LIN {X 0,Y 528.073,Z 998.814,A -85,B 0,C 180,E1 -10169.241,E2 -10169.241} C_VEL
LIN {X 0,Y 528.091,Z 998.55,A -85,B 0,C 180,E1 -10171.628,E2 -10171.628} C_VEL
LIN {X 0,Y 528.095,Z 996.5,A -85,B 0,C 180,E1 -10174.235,E2 -10174.235} C_VEL
LIN {X 0,Y 528.112,Z 993.292,A -85,B 0,C 180,E1 -10176.523,E2 -10176.523} C_VEL
LIN {X 0,Y 528.202,Z 987.95,A -85,B 0,C 180,E1 -10179.15,E2 -10179.15} C_VEL
LIN {X 0,Y 528.409,Z 981.754,A -85,B 0,C 180,E1 -10181.421,E2 -10181.421} C_VEL
LIN {X 0,Y 528.804,Z 973.873,A -85,B 0,C 180,E1 -10183.783,E2 -10183.783} C_VEL
LIN {X 0,Y 529.458,Z 963.843,A -85,B 0,C 180,E1 -10186.23,E2 -10186.23} C_VEL
LIN {X 0,Y 530.258,Z 953.621,A -85,B 0,C 180,E1 -10188.355,E2 -10188.355} C_VEL
LIN {X 0,Y 531.541,Z 939.728,A -85,B 0,C 180,E1 -10190.826,E2 -10190.826} C_VEL
LIN {X 0,Y 532.919,Z 926.263,A -85,B 0,C 180,E1 -10192.891,E2 -10192.891} C_VEL
LIN {X 0,Y 534.753,Z 909.549,A -85,B 0,C 180,E1 -10195.116,E2 -10195.116} C_VEL
LIN {X 0,Y 536.55,Z 894.005,A -85,B 0,C 180,E1 -10196.926,E2 -10196.926} C_VEL
LIN {X 0,Y 538.909,Z 873.935,A -85,B 0,C 180,E1 -10198.964,E2 -10198.964} C_VEL
LIN {X 0,Y 541.194,Z 854.701,A -85,B 0,C 180,E1 -10200.659,E2 -10200.659} C_VEL
LIN {X 0,Y 543.603,Z 833.893,A -85,B 0,C 180,E1 -10202.237,E2 -10202.237} C_VEL
LIN {X 0,Y 545.862,Z 813.459,A -85,B 0,C 180,E1 -10203.586,E2 -10203.586} C_VEL
LIN {X 0,Y 548.077,Z 791.418,A -85,B 0,C 180,E1 -10204.822,E2 -10204.822} C_VEL
LIN {X 0,Y 550.284,Z 768.641,A -85,B 0,C 180,E1 -10205.902,E2 -10205.902} C_VEL
LIN {X 0,Y 552.167,Z 745.38,A -85,B 0,C 180,E1 -10206.794,E2 -10206.794} C_VEL
LIN {X 0,Y 553.867,Z 721.472,A -85,B 0,C 180,E1 -10207.53,E2 -10207.53} C_VEL
LIN {X 0,Y 555.081,Z 698.627,A -85,B 0,C 180,E1 -10208.055,E2 -10208.055} C_VEL
LIN {X 0,Y 556.026,Z 670.252,A -85,B 0,C 180,E1 -10208.516,E2 -10208.516} C_VEL
LIN {X 0,Y 558.703,Z 568.517,A -85,B 0,C 180,E1 -10210.011,E2 -10210.011} C_VEL
LIN {X 0,Y 562.298,Z 475.68,A -85,B 0,C 180,E1 -10211.53,E2 -10211.53} C_VEL
LIN {X 0,Y 567.172,Z 389.799,A -85,B 0,C 180,E1 -10213.068,E2 -10213.068} C_VEL
LIN {X 0,Y 570.884,Z 340.567,A -85,B 0,C 180,E1 -10214.019,E2 -10214.019} C_VEL
LIN {X 0,Y 571.881,Z 338.159,A -85,B 0,C 180,E1 -10214.167,E2 -10214.167} C_VEL
LIN {X 0,Y 579.094,Z 319.344,A -85,B 0,C 180,E1 -10215.771,E2 -10215.771} C_VEL
LIN {X 0,Y 582.937,Z 311.16,A -85,B 0,C 180,E1 -10216.542,E2 -10216.542} C_VEL
LIN {X 0,Y 582.832,Z 309.162,A -85,B 0,C 180,E1 -10217.606,E2 -10217.606} C_VEL
LIN {X 0,Y 582.89,Z 308.585,A -85,B 0,C 180,E1 -10218.273,E2 -10218.273} C_VEL
LIN {X 0,Y 582.338,Z 310.355,A -85,B 0,C 180,E1 -10219.595,E2 -10219.595} C_VEL
LIN {X 0,Y 574.337,Z 326.452,A -85,B 0,C 180,E1 -10221.318,E2 -10221.318} C_VEL
LIN {X 0,Y 566.735,Z 346.819,A -85,B 0,C 180,E1 -10223.329,E2 -10223.329} C_VEL
LIN {X 0,Y 559.494,Z 373.809,A -85,B 0,C 180,E1 -10225.802,E2 -10225.802} C_VEL
LIN {X 0,Y 554.301,Z 400.115,A -85,B 0,C 180,E1 -10228.04,E2 -10228.04} C_VEL
LIN {X 0,Y 555.519,Z 423.333,A -85,B 0,C 180,E1 -10229.307,E2 -10229.307} C_VEL
LIN {X 0,Y 556.922,Z 451.305,A -85,B 0,C 180,E1 -10230.635,E2 -10230.635} C_VEL
LIN {X 0,Y 558.184,Z 484.283,A -85,B 0,C 180,E1 -10231.98,E2 -10231.98} C_VEL
LIN {X 0,Y 558.47,Z 501.799,A -85,B 0,C 180,E1 -10232.6,E2 -10232.6} C_VEL
LIN {X 0,Y 549.884,Z 603.402,A -85,B 0,C 180,E1 -10234.933,E2 -10234.933} C_VEL
LIN {X 0,Y 544.198,Z 689.935,A -85,B 0,C 180,E1 -10236.896,E2 -10236.896} C_VEL
LIN {X 0,Y 542.555,Z 713.994,A -85,B 0,C 180,E1 -10237.66,E2 -10237.66} C_VEL
LIN {X 0,Y 541.005,Z 736.005,A -85,B 0,C 180,E1 -10238.568,E2 -10238.568} C_VEL
LIN {X 0,Y 539.398,Z 756.989,A -85,B 0,C 180,E1 -10239.661,E2 -10239.661} C_VEL
LIN {X 0,Y 538.011,Z 774.87,A -85,B 0,C 180,E1 -10240.795,E2 -10240.795} C_VEL
LIN {X 0,Y 536.611,Z 791.893,A -85,B 0,C 180,E1 -10242.094,E2 -10242.094} C_VEL
LIN {X 0,Y 535.34,Z 806.843,A -85,B 0,C 180,E1 -10243.451,E2 -10243.451} C_VEL
LIN {X 0,Y 534.145,Z 820.367,A -85,B 0,C 180,E1 -10244.918,E2 -10244.918} C_VEL
LIN {X 0,Y 533.023,Z 832.916,A -85,B 0,C 180,E1 -10246.549,E2 -10246.549} C_VEL
LIN {X 0,Y 532.018,Z 843.847,A -85,B 0,C 180,E1 -10248.289,E2 -10248.289} C_VEL
LIN {X 0,Y 531.163,Z 853.18,A -85,B 0,C 180,E1 -10250.136,E2 -10250.136} C_VEL
LIN {X 0,Y 530.507,Z 860.457,A -85,B 0,C 180,E1 -10251.983,E2 -10251.983} C_VEL
LIN {X 0,Y 530,Z 866.128,A -85,B 0,C 180,E1 -10253.935,E2 -10253.935} C_VEL
LIN {X 0,Y 529.624,Z 869.937,A -85,B 0,C 180,E1 -10255.886,E2 -10255.886} C_VEL
LIN {X 0,Y 529.372,Z 871.943,A -85,B 0,C 180,E1 -10257.835,E2 -10257.835} C_VEL
LIN {X 0,Y 529.209,Z 872.179,A -85,B 0,C 180,E1 -10259.892,E2 -10259.892} C_VEL
LIN {X 0,Y 529.126,Z 870.512,A -85,B 0,C 180,E1 -10261.949,E2 -10261.949} C_VEL
LIN {X 0,Y 529.146,Z 867.199,A -85,B 0,C 180,E1 -10263.901,E2 -10263.901} C_VEL
LIN {X 0,Y 529.276,Z 862.125,A -85,B 0,C 180,E1 -10265.855,E2 -10265.855} C_VEL
LIN {X 0,Y 529.52,Z 855.186,A -85,B 0,C 180,E1 -10267.814,E2 -10267.814} C_VEL
LIN {X 0,Y 529.941,Z 846.185,A -85,B 0,C 180,E1 -10269.777,E2 -10269.777} C_VEL
LIN {X 0,Y 530.543,Z 835.567,A -85,B 0,C 180,E1 -10271.634,E2 -10271.634} C_VEL
LIN {X 0,Y 531.311,Z 823.375,A -85,B 0,C 180,E1 -10273.384,E2 -10273.384} C_VEL
LIN {X 0,Y 532.271,Z 809.122,A -85,B 0,C 180,E1 -10275.079,E2 -10275.079} C_VEL
LIN {X 0,Y 533.351,Z 793.597,A -85,B 0,C 180,E1 -10276.613,E2 -10276.613} C_VEL
LIN {X 0,Y 534.503,Z 776.998,A -85,B 0,C 180,E1 -10277.979,E2 -10277.979} C_VEL
LIN {X 0,Y 535.659,Z 759.422,A -85,B 0,C 180,E1 -10279.18,E2 -10279.18} C_VEL
LIN {X 0,Y 536.845,Z 740.956,A -85,B 0,C 180,E1 -10280.212,E2 -10280.212} C_VEL
LIN {X 0,Y 537.985,Z 720.972,A -85,B 0,C 180,E1 -10281.106,E2 -10281.106} C_VEL
LIN {X 0,Y 538.984,Z 700.182,A -85,B 0,C 180,E1 -10281.812,E2 -10281.812} C_VEL
LIN {X 0,Y 539.819,Z 679.295,A -85,B 0,C 180,E1 -10282.316,E2 -10282.316} C_VEL
LIN {X 0,Y 545.343,Z 494.327,A -85,B 0,C 180,E1 -10285.454,E2 -10285.454} C_VEL
LIN {X 0,Y 540.838,Z 450.424,A -85,B 0,C 180,E1 -10286.544,E2 -10286.544} C_VEL
LIN {X 0,Y 544.277,Z 398.054,A -85,B 0,C 180,E1 -10290.14,E2 -10290.14} C_VEL
LIN {X 0,Y 547.874,Z 348.579,A -85,B 0,C 180,E1 -10293.572,E2 -10293.572} C_VEL
LIN {X 0,Y 552.064,Z 296.542,A -85,B 0,C 180,E1 -10297.224,E2 -10297.224} C_VEL
LIN {X 0,Y 553.399,Z 279.163,A -85,B 0,C 180,E1 -10298.468,E2 -10298.468} C_VEL
LIN {X 0,Y 544.537,Z 255.5,A -85,B 0,C 180,E1 -10301.002,E2 -10301.002} C_VEL
LIN {X 0,Y 535.075,Z 232.411,A -85,B 0,C 180,E1 -10303.682,E2 -10303.682} C_VEL
LIN {X 0,Y 534.781,Z 231.7,A -85,B 0,C 180,E1 -10303.773,E2 -10303.773} C_VEL
LIN {X 0,Y 536.691,Z 232.864,A -85,B 0,C 180,E1 -10304.059,E2 -10304.059} C_VEL
LIN {X 0,Y 546.06,Z 252.219,A -85,B 0,C 180,E1 -10306.403,E2 -10306.403} C_VEL
LIN {X 0,Y 554.586,Z 272.537,A -85,B 0,C 180,E1 -10308.749,E2 -10308.749} C_VEL
LIN {X 0,Y 561.348,Z 291.078,A -85,B 0,C 180,E1 -10310.79,E2 -10310.79} C_VEL
LIN {X 0,Y 561.17,Z 298.745,A -85,B 0,C 180,E1 -10311.342,E2 -10311.342} C_VEL
LIN {X 0,Y 560.235,Z 305.401,A -85,B 0,C 180,E1 -10311.739,E2 -10311.739} C_VEL
LIN {X 0,Y 555.035,Z 324.312,A -85,B 0,C 180,E1 -10312.584,E2 -10312.584} C_VEL
LIN {X 0,Y 554.398,Z 330.093,A -85,B 0,C 180,E1 -10312.919,E2 -10312.919} C_VEL
LIN {X 0,Y 554.416,Z 348.963,A -85,B 0,C 180,E1 -10314.148,E2 -10314.148} C_VEL
LIN {X 0,Y 552.164,Z 359.982,A -85,B 0,C 180,E1 -10314.558,E2 -10314.558} C_VEL
LIN {X 0,Y 549.54,Z 449.417,A -85,B 0,C 180,E1 -10315.862,E2 -10315.862} C_VEL
LIN {X 0,Y 546.257,Z 527.382,A -85,B 0,C 180,E1 -10317.185,E2 -10317.185} C_VEL
LIN {X 0,Y 541.758,Z 616.567,A -85,B 0,C 180,E1 -10318.913,E2 -10318.913} C_VEL
LIN {X 0,Y 540.542,Z 646.224,A -85,B 0,C 180,E1 -10319.6,E2 -10319.6} C_VEL
LIN {X 0,Y 539.38,Z 668.071,A -85,B 0,C 180,E1 -10320.302,E2 -10320.302} C_VEL
LIN {X 0,Y 537.858,Z 689.945,A -85,B 0,C 180,E1 -10321.217,E2 -10321.217} C_VEL
LIN {X 0,Y 536.147,Z 710.107,A -85,B 0,C 180,E1 -10322.27,E2 -10322.27} C_VEL
LIN {X 0,Y 534.288,Z 729.488,A -85,B 0,C 180,E1 -10323.491,E2 -10323.491} C_VEL
LIN {X 0,Y 532.25,Z 748.721,A -85,B 0,C 180,E1 -10324.936,E2 -10324.936} C_VEL
LIN {X 0,Y 530.139,Z 767.337,A -85,B 0,C 180,E1 -10326.597,E2 -10326.597} C_VEL
LIN {X 0,Y 528.194,Z 784.001,A -85,B 0,C 180,E1 -10328.355,E2 -10328.355} C_VEL
LIN {X 0,Y 526.509,Z 798.406,A -85,B 0,C 180,E1 -10330.127,E2 -10330.127} C_VEL
LIN {X 0,Y 524.913,Z 812.343,A -85,B 0,C 180,E1 -10332.14,E2 -10332.14} C_VEL
LIN {X 0,Y 523.561,Z 824.713,A -85,B 0,C 180,E1 -10334.268,E2 -10334.268} C_VEL
LIN {X 0,Y 522.516,Z 835.264,A -85,B 0,C 180,E1 -10336.438,E2 -10336.438} C_VEL
LIN {X 0,Y 521.742,Z 844.408,A -85,B 0,C 180,E1 -10338.727,E2 -10338.727} C_VEL
LIN {X 0,Y 521.227,Z 851.534,A -85,B 0,C 180,E1 -10340.949,E2 -10340.949} C_VEL
LIN {X 0,Y 520.916,Z 857.237,A -85,B 0,C 180,E1 -10343.276,E2 -10343.276} C_VEL
LIN {X 0,Y 520.738,Z 861.151,A -85,B 0,C 180,E1 -10345.595,E2 -10345.595} C_VEL
LIN {X 0,Y 520.657,Z 863.456,A -85,B 0,C 180,E1 -10347.909,E2 -10347.909} C_VEL
LIN {X 0,Y 520.639,Z 864.185,A -85,B 0,C 180,E1 -10350.22,E2 -10350.22} C_VEL
LIN {X 0,Y 520.658,Z 863.243,A -85,B 0,C 180,E1 -10352.532,E2 -10352.532} C_VEL
LIN {X 0,Y 520.758,Z 860.648,A -85,B 0,C 180,E1 -10354.846,E2 -10354.846} C_VEL
LIN {X 0,Y 520.942,Z 856.196,A -85,B 0,C 180,E1 -10357.278,E2 -10357.278} C_VEL
LIN {X 0,Y 521.293,Z 850.544,A -85,B 0,C 180,E1 -10359.495,E2 -10359.495} C_VEL
LIN {X 0,Y 521.889,Z 842.757,A -85,B 0,C 180,E1 -10361.83,E2 -10361.83} C_VEL
LIN {X 0,Y 522.691,Z 833.442,A -85,B 0,C 180,E1 -10364.06,E2 -10364.06} C_VEL
LIN {X 0,Y 523.79,Z 822.558,A -85,B 0,C 180,E1 -10366.217,E2 -10366.217} C_VEL
LIN {X 0,Y 525.167,Z 809.983,A -85,B 0,C 180,E1 -10368.31,E2 -10368.31} C_VEL
LIN {X 0,Y 526.732,Z 796.54,A -85,B 0,C 180,E1 -10370.212,E2 -10370.212} C_VEL
LIN {X 0,Y 528.506,Z 781.567,A -85,B 0,C 180,E1 -10372.021,E2 -10372.021} C_VEL
LIN {X 0,Y 530.475,Z 764.694,A -85,B 0,C 180,E1 -10373.753,E2 -10373.753} C_VEL
LIN {X 0,Y 532.444,Z 747.087,A -85,B 0,C 180,E1 -10375.292,E2 -10375.292} C_VEL
LIN {X 0,Y 534.424,Z 728.325,A -85,B 0,C 180,E1 -10376.682,E2 -10376.682} C_VEL
LIN {X 0,Y 536.282,Z 708.692,A -85,B 0,C 180,E1 -10377.904,E2 -10377.904} C_VEL
LIN {X 0,Y 537.972,Z 688.594,A -85,B 0,C 180,E1 -10378.938,E2 -10378.938} C_VEL
LIN {X 0,Y 539.445,Z 667.47,A -85,B 0,C 180,E1 -10379.815,E2 -10379.815} C_VEL
LIN {X 0,Y 540.613,Z 645.234,A -85,B 0,C 180,E1 -10380.523,E2 -10380.523} C_VEL
LIN {X 0,Y 541.962,Z 612.731,A -85,B 0,C 180,E1 -10381.262,E2 -10381.262} C_VEL
LIN {X 0,Y 546.474,Z 523.52,A -85,B 0,C 180,E1 -10382.98,E2 -10382.98} C_VEL
LIN {X 0,Y 549.681,Z 446.416,A -85,B 0,C 180,E1 -10384.279,E2 -10384.279} C_VEL
LIN {X 0,Y 552.294,Z 358.711,A -85,B 0,C 180,E1 -10385.563,E2 -10385.563} C_VEL
LIN {X 0,Y 554.559,Z 348.099,A -85,B 0,C 180,E1 -10386,E2 -10386} C_VEL
LIN {X 0,Y 554.663,Z 312.521,A -85,B 0,C 180,E1 -10388.391,E2 -10388.391} C_VEL
LIN {X 0,Y 554.973,Z 294.272,A -85,B 0,C 180,E1 -10389.707,E2 -10389.707} C_VEL
LIN {X 0,Y 547.767,Z 275.074,A -85,B 0,C 180,E1 -10391.861,E2 -10391.861} C_VEL
LIN {X 0,Y 539.853,Z 256.334,A -85,B 0,C 180,E1 -10394.058,E2 -10394.058} C_VEL
LIN {X 0,Y 532.349,Z 240.84,A -85,B 0,C 180,E1 -10395.976,E2 -10395.976} C_VEL
LIN {X 0,Y 526.336,Z 229.281,A -85,B 0,C 180,E1 -10397.445,E2 -10397.445} C_VEL
LIN {X 0,Y 523.694,Z 224.562,A -85,B 0,C 180,E1 -10398.067,E2 -10398.067} C_VEL
LIN {X 0,Y 521.964,Z 221.334,A -85,B 0,C 180,E1 -10398.485,E2 -10398.485} C_VEL
LIN {X 0,Y 521.744,Z 220.235,A -85,B 0,C 180,E1 -10398.61,E2 -10398.61} C_VEL
LIN {X 0,Y 521.743,Z 220.233,A -85,B 0,C 180,E1 -10402.035,E2 -10402.035} C_VEL
LIN {X 0,Y 521.737,Z 220.239,A -85,B 0,C 180,E1 -10405.495,E2 -10405.495} C_VEL
LIN {X 0,Y 521.735,Z 220.239,A -85,B 0,C 180,E1 -10408.967,E2 -10408.967} C_VEL
LIN {X 0,Y 521.739,Z 220.219,A -85,B 0,C 180,E1 -10412.368,E2 -10412.368} C_VEL
LIN {X 0,Y 521.742,Z 220.211,A -85,B 0,C 180,E1 -10415.815,E2 -10415.815} C_VEL
LIN {X 0,Y 521.737,Z 220.238,A -85,B 0,C 180,E1 -10419.266,E2 -10419.266} C_VEL
LIN {X 0,Y 521.741,Z 220.21,A -85,B 0,C 180,E1 -10422.719,E2 -10422.719} C_VEL
LIN {X 0,Y 521.732,Z 220.223,A -85,B 0,C 180,E1 -10426.139,E2 -10426.139} C_VEL
LIN {X 0,Y 521.742,Z 220.225,A -85,B 0,C 180,E1 -10429.622,E2 -10429.622} C_VEL
LIN {X 0,Y 521.745,Z 220.21,A -85,B 0,C 180,E1 -10433.078,E2 -10433.078} C_VEL
LIN {X 0,Y 521.729,Z 220.239,A -85,B 0,C 180,E1 -10436.594,E2 -10436.594} C_VEL
LIN {X 0,Y 521.726,Z 220.202,A -85,B 0,C 180,E1 -10440.11,E2 -10440.11} C_VEL
LIN {X 0,Y 521.744,Z 220.238,A -85,B 0,C 180,E1 -10443.516,E2 -10443.516} C_VEL
LIN {X 0,Y 521.744,Z 220.198,A -85,B 0,C 180,E1 -10447.045,E2 -10447.045} C_VEL
LIN {X 0,Y 521.72,Z 220.241,A -85,B 0,C 180,E1 -10450.524,E2 -10450.524} C_VEL
LIN {X 0,Y 521.739,Z 220.242,A -85,B 0,C 180,E1 -10453.974,E2 -10453.974} C_VEL
LIN {X 0,Y 521.749,Z 220.241,A -85,B 0,C 180,E1 -10457.395,E2 -10457.395} C_VEL
LIN {X 0,Y 521.717,Z 220.239,A -85,B 0,C 180,E1 -10460.767,E2 -10460.767} C_VEL
LIN {X 0,Y 521.722,Z 220.235,A -85,B 0,C 180,E1 -10464.213,E2 -10464.213} C_VEL
LIN {X 0,Y 521.753,Z 220.235,A -85,B 0,C 180,E1 -10467.631,E2 -10467.631} C_VEL
LIN {X 0,Y 521.722,Z 220.239,A -85,B 0,C 180,E1 -10471.054,E2 -10471.054} C_VEL
LIN {X 0,Y 521.754,Z 220.325,A -85,B 0,C 180,E1 -10473.388,E2 -10473.388} C_VEL
LIN {X 0,Y 522.874,Z 223.439,A -85,B 0,C 180,E1 -10473.813,E2 -10473.813} C_VEL
LIN {X 0,Y 524.045,Z 225.27,A -85,B 0,C 180,E1 -10474.122,E2 -10474.122} C_VEL
LIN {X 0,Y 525.794,Z 228.852,A -85,B 0,C 180,E1 -10474.653,E2 -10474.653} C_VEL
LIN {X 0,Y 533.823,Z 244.524,A -85,B 0,C 180,E1 -10476.96,E2 -10476.96} C_VEL
LIN {X 0,Y 543.759,Z 264.219,A -85,B 0,C 180,E1 -10479.649,E2 -10479.649} C_VEL
LIN {X 0,Y 556.286,Z 289.963,A -85,B 0,C 180,E1 -10482.832,E2 -10482.832} C_VEL
LIN {X 0,Y 561.303,Z 300.628,A -85,B 0,C 180,E1 -10484.054,E2 -10484.054} C_VEL
LIN {X 0,Y 559.967,Z 313.808,A -85,B 0,C 180,E1 -10484.827,E2 -10484.827} C_VEL
LIN {X 0,Y 562.81,Z 340.382,A -85,B 0,C 180,E1 -10485.543,E2 -10485.543} C_VEL
LIN {X 0,Y 554.944,Z 572.433,A -85,B 0,C 180,E1 -10489.082,E2 -10489.082} C_VEL
LIN {X 0,Y 551.384,Z 692.781,A -85,B 0,C 180,E1 -10490.881,E2 -10490.881} C_VEL
LIN {X 0,Y 549.935,Z 717.309,A -85,B 0,C 180,E1 -10491.421,E2 -10491.421} C_VEL
LIN {X 0,Y 548.22,Z 740.807,A -85,B 0,C 180,E1 -10492.107,E2 -10492.107} C_VEL
LIN {X 0,Y 546.127,Z 763.625,A -85,B 0,C 180,E1 -10492.965,E2 -10492.965} C_VEL
LIN {X 0,Y 543.758,Z 786.648,A -85,B 0,C 180,E1 -10494.008,E2 -10494.008} C_VEL
LIN {X 0,Y 541.136,Z 809.081,A -85,B 0,C 180,E1 -10495.247,E2 -10495.247} C_VEL
LIN {X 0,Y 538.432,Z 830.883,A -85,B 0,C 180,E1 -10496.655,E2 -10496.655} C_VEL
LIN {X 0,Y 535.859,Z 850.246,A -85,B 0,C 180,E1 -10498.125,E2 -10498.125} C_VEL
LIN {X 0,Y 533.106,Z 870.475,A -85,B 0,C 180,E1 -10499.886,E2 -10499.886} C_VEL
LIN {X 0,Y 530.656,Z 888,A -85,B 0,C 180,E1 -10501.652,E2 -10501.652} C_VEL
LIN {X 0,Y 528.37,Z 904.978,A -85,B 0,C 180,E1 -10503.595,E2 -10503.595} C_VEL
LIN {X 0,Y 526.295,Z 920.525,A -85,B 0,C 180,E1 -10505.652,E2 -10505.652} C_VEL
LIN {X 0,Y 524.481,Z 935.456,A -85,B 0,C 180,E1 -10507.901,E2 -10507.901} C_VEL
LIN {X 0,Y 523.037,Z 948.215,A -85,B 0,C 180,E1 -10510.146,E2 -10510.146} C_VEL
LIN {X 0,Y 521.869,Z 960.375,A -85,B 0,C 180,E1 -10512.609,E2 -10512.609} C_VEL
LIN {X 0,Y 521.085,Z 970.191,A -85,B 0,C 180,E1 -10514.987,E2 -10514.987} C_VEL
LIN {X 0,Y 520.553,Z 978.856,A -85,B 0,C 180,E1 -10517.464,E2 -10517.464} C_VEL
LIN {X 0,Y 520.257,Z 985.967,A -85,B 0,C 180,E1 -10520.039,E2 -10520.039} C_VEL
LIN {X 0,Y 520.116,Z 990.812,A -85,B 0,C 180,E1 -10522.266,E2 -10522.266} C_VEL
LIN {X 0,Y 520.085,Z 994.867,A -85,B 0,C 180,E1 -10524.816,E2 -10524.816} C_VEL
LIN {X 0,Y 520.101,Z 997.064,A -85,B 0,C 180,E1 -10527.135,E2 -10527.135} C_VEL
LIN {X 0,Y 520.12,Z 997.946,A -85,B 0,C 180,E1 -10529.229,E2 -10529.229} C_VEL
LIN {X 0,Y 520.139,Z 997.696,A -85,B 0,C 180,E1 -10531.561,E2 -10531.561} C_VEL
LIN {X 0,Y 520.139,Z 995.709,A -85,B 0,C 180,E1 -10534.189,E2 -10534.189} C_VEL
LIN {X 0,Y 520.149,Z 992.525,A -85,B 0,C 180,E1 -10536.512,E2 -10536.512} C_VEL
LIN {X 0,Y 520.233,Z 987.22,A -85,B 0,C 180,E1 -10539.18,E2 -10539.18} C_VEL
LIN {X 0,Y 520.439,Z 980.92,A -85,B 0,C 180,E1 -10541.526,E2 -10541.526} C_VEL
LIN {X 0,Y 520.81,Z 973.556,A -85,B 0,C 180,E1 -10543.772,E2 -10543.772} C_VEL
LIN {X 0,Y 521.5,Z 963.155,A -85,B 0,C 180,E1 -10546.371,E2 -10546.371} C_VEL
LIN {X 0,Y 522.274,Z 953.521,A -85,B 0,C 180,E1 -10548.415,E2 -10548.415} C_VEL
LIN {X 0,Y 523.524,Z 940.476,A -85,B 0,C 180,E1 -10550.809,E2 -10550.809} C_VEL
LIN {X 0,Y 524.882,Z 927.409,A -85,B 0,C 180,E1 -10552.869,E2 -10552.869} C_VEL
LIN {X 0,Y 526.69,Z 911.753,A -85,B 0,C 180,E1 -10555.047,E2 -10555.047} C_VEL
LIN {X 0,Y 528.751,Z 894.474,A -85,B 0,C 180,E1 -10557.113,E2 -10557.113} C_VEL
LIN {X 0,Y 531.057,Z 875.875,A -85,B 0,C 180,E1 -10559.063,E2 -10559.063} C_VEL
LIN {X 0,Y 533.395,Z 856.932,A -85,B 0,C 180,E1 -10560.781,E2 -10560.781} C_VEL
LIN {X 0,Y 536.068,Z 835.167,A -85,B 0,C 180,E1 -10562.492,E2 -10562.492} C_VEL
LIN {X 0,Y 538.313,Z 815.895,A -85,B 0,C 180,E1 -10563.801,E2 -10563.801} C_VEL
LIN {X 0,Y 540.838,Z 792.483,A -85,B 0,C 180,E1 -10565.162,E2 -10565.162} C_VEL
LIN {X 0,Y 543.143,Z 769.878,A -85,B 0,C 180,E1 -10566.261,E2 -10566.261} C_VEL
LIN {X 0,Y 545.171,Z 746.679,A -85,B 0,C 180,E1 -10567.181,E2 -10567.181} C_VEL
LIN {X 0,Y 546.946,Z 723.653,A -85,B 0,C 180,E1 -10567.919,E2 -10567.919} C_VEL
LIN {X 0,Y 548.337,Z 699.785,A -85,B 0,C 180,E1 -10568.49,E2 -10568.49} C_VEL
LIN {X 0,Y 549.321,Z 674.5,A -85,B 0,C 180,E1 -10568.926,E2 -10568.926} C_VEL
LIN {X 0,Y 552.201,Z 576.067,A -85,B 0,C 180,E1 -10570.412,E2 -10570.412} C_VEL
LIN {X 0,Y 556.018,Z 486.791,A -85,B 0,C 180,E1 -10571.912,E2 -10571.912} C_VEL
LIN {X 0,Y 561.161,Z 403.595,A -85,B 0,C 180,E1 -10573.442,E2 -10573.442} C_VEL
LIN {X 0,Y 566.111,Z 343.623,A -85,B 0,C 180,E1 -10574.63,E2 -10574.63} C_VEL
LIN {X 0,Y 567.547,Z 340.563,A -85,B 0,C 180,E1 -10574.806,E2 -10574.806} C_VEL
LIN {X 0,Y 575.021,Z 323.124,A -85,B 0,C 180,E1 -10576.343,E2 -10576.343} C_VEL
LIN {X 0,Y 578.257,Z 316.88,A -85,B 0,C 180,E1 -10576.934,E2 -10576.934} C_VEL
LIN {X 0,Y 578.346,Z 315.09,A -85,B 0,C 180,E1 -10578.172,E2 -10578.172} C_VEL
LIN {X 0,Y 577.731,Z 316.371,A -85,B 0,C 180,E1 -10579.238,E2 -10579.238} C_VEL
LIN {X 0,Y 568.969,Z 332.766,A -85,B 0,C 180,E1 -10581.013,E2 -10581.013} C_VEL
LIN {X 0,Y 561.23,Z 352.221,A -85,B 0,C 180,E1 -10582.973,E2 -10582.973} C_VEL
LIN {X 0,Y 553.999,Z 376.806,A -85,B 0,C 180,E1 -10585.289,E2 -10585.289} C_VEL
LIN {X 0,Y 549.797,Z 396.074,A -85,B 0,C 180,E1 -10586.972,E2 -10586.972} C_VEL
LIN {X 0,Y 550.632,Z 420.862,A -85,B 0,C 180,E1 -10588.423,E2 -10588.423} C_VEL
LIN {X 0,Y 551.732,Z 450.81,A -85,B 0,C 180,E1 -10589.92,E2 -10589.92} C_VEL
LIN {X 0,Y 552.582,Z 483.66,A -85,B 0,C 180,E1 -10591.317,E2 -10591.317} C_VEL
LIN {X 0,Y 552.788,Z 503.004,A -85,B 0,C 180,E1 -10592.031,E2 -10592.031} C_VEL
LIN {X 0,Y 543.196,Z 609.107,A -85,B 0,C 180,E1 -10594.537,E2 -10594.537} C_VEL
LIN {X 0,Y 537.537,Z 689.387,A -85,B 0,C 180,E1 -10596.414,E2 -10596.414} C_VEL
LIN {X 0,Y 535.83,Z 712.83,A -85,B 0,C 180,E1 -10597.161,E2 -10597.161} C_VEL
LIN {X 0,Y 534.14,Z 734.712,A -85,B 0,C 180,E1 -10598.071,E2 -10598.071} C_VEL
LIN {X 0,Y 532.54,Z 754.757,A -85,B 0,C 180,E1 -10599.1,E2 -10599.1} C_VEL
LIN {X 0,Y 530.937,Z 773.824,A -85,B 0,C 180,E1 -10600.299,E2 -10600.299} C_VEL
LIN {X 0,Y 529.443,Z 791.217,A -85,B 0,C 180,E1 -10601.615,E2 -10601.615} C_VEL
LIN {X 0,Y 527.95,Z 807.44,A -85,B 0,C 180,E1 -10603.099,E2 -10603.099} C_VEL
LIN {X 0,Y 526.676,Z 821.085,A -85,B 0,C 180,E1 -10604.586,E2 -10604.586} C_VEL
LIN {X 0,Y 525.456,Z 833.65,A -85,B 0,C 180,E1 -10606.24,E2 -10606.24} C_VEL
LIN {X 0,Y 524.372,Z 844.771,A -85,B 0,C 180,E1 -10608.017,E2 -10608.017} C_VEL
LIN {X 0,Y 523.445,Z 854.084,A -85,B 0,C 180,E1 -10609.878,E2 -10609.878} C_VEL
LIN {X 0,Y 522.727,Z 861.417,A -85,B 0,C 180,E1 -10611.752,E2 -10611.752} C_VEL
LIN {X 0,Y 522.168,Z 867.158,A -85,B 0,C 180,E1 -10613.734,E2 -10613.734} C_VEL
LIN {X 0,Y 521.752,Z 870.983,A -85,B 0,C 180,E1 -10615.714,E2 -10615.714} C_VEL
LIN {X 0,Y 521.458,Z 873.086,A -85,B 0,C 180,E1 -10617.802,E2 -10617.802} C_VEL
LIN {X 0,Y 521.288,Z 873.282,A -85,B 0,C 180,E1 -10619.78,E2 -10619.78} C_VEL
LIN {X 0,Y 521.191,Z 871.638,A -85,B 0,C 180,E1 -10621.869,E2 -10621.869} C_VEL
LIN {X 0,Y 521.209,Z 868.088,A -85,B 0,C 180,E1 -10623.96,E2 -10623.96} C_VEL
LIN {X 0,Y 521.345,Z 862.924,A -85,B 0,C 180,E1 -10625.945,E2 -10625.945} C_VEL
LIN {X 0,Y 521.604,Z 855.883,A -85,B 0,C 180,E1 -10627.933,E2 -10627.933} C_VEL
LIN {X 0,Y 522.02,Z 847.345,A -85,B 0,C 180,E1 -10629.815,E2 -10629.815} C_VEL
LIN {X 0,Y 522.64,Z 836.731,A -85,B 0,C 180,E1 -10631.7,E2 -10631.7} C_VEL
LIN {X 0,Y 523.432,Z 824.547,A -85,B 0,C 180,E1 -10633.477,E2 -10633.477} C_VEL
LIN {X 0,Y 524.389,Z 810.796,A -85,B 0,C 180,E1 -10635.143,E2 -10635.143} C_VEL
LIN {X 0,Y 525.493,Z 795.428,A -85,B 0,C 180,E1 -10636.698,E2 -10636.698} C_VEL
LIN {X 0,Y 526.724,Z 778.299,A -85,B 0,C 180,E1 -10638.139,E2 -10638.139} C_VEL
LIN {X 0,Y 527.917,Z 760.842,A -85,B 0,C 180,E1 -10639.357,E2 -10639.357} C_VEL
LIN {X 0,Y 529.12,Z 742.725,A -85,B 0,C 180,E1 -10640.396,E2 -10640.396} C_VEL
LIN {X 0,Y 530.265,Z 723.546,A -85,B 0,C 180,E1 -10641.284,E2 -10641.284} C_VEL
LIN {X 0,Y 531.332,Z 702.865,A -85,B 0,C 180,E1 -10642.026,E2 -10642.026} C_VEL
LIN {X 0,Y 532.259,Z 681.478,A -85,B 0,C 180,E1 -10642.574,E2 -10642.574} C_VEL
LIN {X 0,Y 538.097,Z 495.341,A -85,B 0,C 180,E1 -10645.799,E2 -10645.799} C_VEL
LIN {X 0,Y 533.475,Z 449.88,A -85,B 0,C 180,E1 -10646.941,E2 -10646.941} C_VEL
LIN {X 0,Y 537.156,Z 396.261,A -85,B 0,C 180,E1 -10650.667,E2 -10650.667} C_VEL
LIN {X 0,Y 540.798,Z 348.675,A -85,B 0,C 180,E1 -10654.007,E2 -10654.007} C_VEL
LIN {X 0,Y 545.201,Z 296.528,A -85,B 0,C 180,E1 -10657.708,E2 -10657.708} C_VEL
LIN {X 0,Y 546.276,Z 282.025,A -85,B 0,C 180,E1 -10658.763,E2 -10658.763} C_VEL
LIN {X 0,Y 537.787,Z 259.311,A -85,B 0,C 180,E1 -10661.229,E2 -10661.229} C_VEL
LIN {X 0,Y 529.445,Z 238.662,A -85,B 0,C 180,E1 -10663.659,E2 -10663.659} C_VEL
LIN {X 0,Y 531.632,Z 239.348,A -85,B 0,C 180,E1 -10663.949,E2 -10663.949} C_VEL
LIN {X 0,Y 539.955,Z 256.58,A -85,B 0,C 180,E1 -10666.084,E2 -10666.084} C_VEL
LIN {X 0,Y 547.54,Z 274.698,A -85,B 0,C 180,E1 -10668.199,E2 -10668.199} C_VEL
LIN {X 0,Y 554.992,Z 294.722,A -85,B 0,C 180,E1 -10670.441,E2 -10670.441} C_VEL
LIN {X 0,Y 554.398,Z 330.093,A -85,B 0,C 180,E1 -10672.919,E2 -10672.919} C_VEL
LIN {X 0,Y 553.581,Z 335.341,A -85,B 0,C 180,E1 -10673.19,E2 -10673.19} C_VEL
LIN {X 0,Y 547.836,Z 351.92,A -85,B 0,C 180,E1 -10673.701,E2 -10673.701} C_VEL
LIN {X 0,Y 545.655,Z 362.546,A -85,B 0,C 180,E1 -10674.097,E2 -10674.097} C_VEL
LIN {X 0,Y 542.944,Z 451.442,A -85,B 0,C 180,E1 -10675.405,E2 -10675.405} C_VEL
LIN {X 0,Y 539.626,Z 527.403,A -85,B 0,C 180,E1 -10676.711,E2 -10676.711} C_VEL
LIN {X 0,Y 535.005,Z 615.09,A -85,B 0,C 180,E1 -10678.434,E2 -10678.434} C_VEL
LIN {X 0,Y 533.624,Z 647.175,A -85,B 0,C 180,E1 -10679.183,E2 -10679.183} C_VEL
LIN {X 0,Y 532.402,Z 669.345,A -85,B 0,C 180,E1 -10679.904,E2 -10679.904} C_VEL
LIN {X 0,Y 530.865,Z 690.529,A -85,B 0,C 180,E1 -10680.802,E2 -10680.802} C_VEL
LIN {X 0,Y 529.086,Z 710.813,A -85,B 0,C 180,E1 -10681.867,E2 -10681.867} C_VEL
LIN {X 0,Y 527.153,Z 730.268,A -85,B 0,C 180,E1 -10683.103,E2 -10683.103} C_VEL
LIN {X 0,Y 525.02,Z 749.549,A -85,B 0,C 180,E1 -10684.567,E2 -10684.567} C_VEL
LIN {X 0,Y 522.942,Z 767.166,A -85,B 0,C 180,E1 -10686.146,E2 -10686.146} C_VEL
LIN {X 0,Y 521.033,Z 782.83,A -85,B 0,C 180,E1 -10687.787,E2 -10687.787} C_VEL
LIN {X 0,Y 519.068,Z 798.679,A -85,B 0,C 180,E1 -10689.739,E2 -10689.739} C_VEL
LIN {X 0,Y 517.376,Z 812.519,A -85,B 0,C 180,E1 -10691.755,E2 -10691.755} C_VEL
LIN {X 0,Y 515.997,Z 824.407,A -85,B 0,C 180,E1 -10693.797,E2 -10693.797} C_VEL
LIN {X 0,Y 514.817,Z 835.488,A -85,B 0,C 180,E1 -10696.064,E2 -10696.064} C_VEL
LIN {X 0,Y 513.987,Z 844.588,A -85,B 0,C 180,E1 -10698.327,E2 -10698.327} C_VEL
LIN {X 0,Y 513.4,Z 851.915,A -85,B 0,C 180,E1 -10700.584,E2 -10700.584} C_VEL
LIN {X 0,Y 513.02,Z 857.723,A -85,B 0,C 180,E1 -10702.947,E2 -10702.947} C_VEL
LIN {X 0,Y 512.827,Z 861.83,A -85,B 0,C 180,E1 -10705.303,E2 -10705.303} C_VEL
LIN {X 0,Y 512.724,Z 864.323,A -85,B 0,C 180,E1 -10707.653,E2 -10707.653} C_VEL
LIN {X 0,Y 512.715,Z 865.211,A -85,B 0,C 180,E1 -10710,E2 -10710} C_VEL
LIN {X 0,Y 512.721,Z 864.377,A -85,B 0,C 180,E1 -10712.347,E2 -10712.347} C_VEL
LIN {X 0,Y 512.823,Z 861.957,A -85,B 0,C 180,E1 -10714.697,E2 -10714.697} C_VEL
LIN {X 0,Y 513.013,Z 857.929,A -85,B 0,C 180,E1 -10717.053,E2 -10717.053} C_VEL
LIN {X 0,Y 513.376,Z 852.172,A -85,B 0,C 180,E1 -10719.416,E2 -10719.416} C_VEL
LIN {X 0,Y 513.959,Z 844.91,A -85,B 0,C 180,E1 -10721.673,E2 -10721.673} C_VEL
LIN {X 0,Y 514.778,Z 835.896,A -85,B 0,C 180,E1 -10723.937,E2 -10723.937} C_VEL
LIN {X 0,Y 515.881,Z 825.52,A -85,B 0,C 180,E1 -10726.091,E2 -10726.091} C_VEL
LIN {X 0,Y 517.236,Z 813.852,A -85,B 0,C 180,E1 -10728.134,E2 -10728.134} C_VEL
LIN {X 0,Y 518.962,Z 799.602,A -85,B 0,C 180,E1 -10730.23,E2 -10730.23} C_VEL
LIN {X 0,Y 520.817,Z 784.56,A -85,B 0,C 180,E1 -10732.104,E2 -10732.104} C_VEL
LIN {X 0,Y 522.772,Z 768.635,A -85,B 0,C 180,E1 -10733.802,E2 -10733.802} C_VEL
LIN {X 0,Y 524.953,Z 750.305,A -85,B 0,C 180,E1 -10735.465,E2 -10735.465} C_VEL
LIN {X 0,Y 527.06,Z 731.305,A -85,B 0,C 180,E1 -10736.919,E2 -10736.919} C_VEL
LIN {X 0,Y 528.977,Z 712.359,A -85,B 0,C 180,E1 -10738.139,E2 -10738.139} C_VEL
LIN {X 0,Y 530.751,Z 692.432,A -85,B 0,C 180,E1 -10739.205,E2 -10739.205} C_VEL
LIN {X 0,Y 532.312,Z 670.851,A -85,B 0,C 180,E1 -10740.132,E2 -10740.132} C_VEL
LIN {X 0,Y 533.516,Z 649.724,A -85,B 0,C 180,E1 -10740.836,E2 -10740.836} C_VEL
LIN {X 0,Y 534.659,Z 622.529,A -85,B 0,C 180,E1 -10741.501,E2 -10741.501} C_VEL
LIN {X 0,Y 539.133,Z 537.667,A -85,B 0,C 180,E1 -10743.193,E2 -10743.193} C_VEL
LIN {X 0,Y 542.511,Z 463.41,A -85,B 0,C 180,E1 -10744.496,E2 -10744.496} C_VEL
LIN {X 0,Y 544.936,Z 390.36,A -85,B 0,C 180,E1 -10745.604,E2 -10745.604} C_VEL
LIN {X 0,Y 545.777,Z 361.482,A -85,B 0,C 180,E1 -10746.021,E2 -10746.021} C_VEL
LIN {X 0,Y 548.279,Z 350.09,A -85,B 0,C 180,E1 -10746.479,E2 -10746.479} C_VEL
LIN {X 0,Y 548.418,Z 314.014,A -85,B 0,C 180,E1 -10748.91,E2 -10748.91} C_VEL
LIN {X 0,Y 548.648,Z 298.086,A -85,B 0,C 180,E1 -10750.054,E2 -10750.054} C_VEL
LIN {X 0,Y 541.116,Z 277.916,A -85,B 0,C 180,E1 -10752.342,E2 -10752.342} C_VEL
LIN {X 0,Y 533.24,Z 259.389,A -85,B 0,C 180,E1 -10754.557,E2 -10754.557} C_VEL
LIN {X 0,Y 524.905,Z 242.374,A -85,B 0,C 180,E1 -10756.704,E2 -10756.704} C_VEL
LIN {X 0,Y 518.482,Z 230.32,A -85,B 0,C 180,E1 -10758.292,E2 -10758.292} C_VEL
LIN {X 0,Y 515.867,Z 225.675,A -85,B 0,C 180,E1 -10758.923,E2 -10758.923} C_VEL
LIN {X 0,Y 514.115,Z 222.681,A -85,B 0,C 180,E1 -10759.342,E2 -10759.342} C_VEL
LIN {X 0,Y 513.798,Z 221.214,A -85,B 0,C 180,E1 -10759.502,E2 -10759.502} C_VEL
LIN {X 0,Y 513.791,Z 221.21,A -85,B 0,C 180,E1 -10763.033,E2 -10763.033} C_VEL
LIN {X 0,Y 513.805,Z 221.208,A -85,B 0,C 180,E1 -10766.449,E2 -10766.449} C_VEL
LIN {X 0,Y 513.805,Z 221.222,A -85,B 0,C 180,E1 -10769.996,E2 -10769.996} C_VEL
LIN {X 0,Y 513.798,Z 221.224,A -85,B 0,C 180,E1 -10773.41,E2 -10773.41} C_VEL
LIN {X 0,Y 513.8,Z 221.196,A -85,B 0,C 180,E1 -10776.998,E2 -10776.998} C_VEL
LIN {X 0,Y 513.797,Z 221.214,A -85,B 0,C 180,E1 -10780.444,E2 -10780.444} C_VEL
LIN {X 0,Y 513.8,Z 221.221,A -85,B 0,C 180,E1 -10784.02,E2 -10784.02} C_VEL
LIN {X 0,Y 513.797,Z 221.192,A -85,B 0,C 180,E1 -10787.411,E2 -10787.411} C_VEL
LIN {X 0,Y 513.806,Z 221.226,A -85,B 0,C 180,E1 -10790.931,E2 -10790.931} C_VEL
LIN {X 0,Y 513.785,Z 221.192,A -85,B 0,C 180,E1 -10794.416,E2 -10794.416} C_VEL
LIN {X 0,Y 513.802,Z 221.226,A -85,B 0,C 180,E1 -10797.881,E2 -10797.881} C_VEL
LIN {X 0,Y 513.802,Z 221.191,A -85,B 0,C 180,E1 -10801.338,E2 -10801.338} C_VEL
LIN {X 0,Y 513.795,Z 221.224,A -85,B 0,C 180,E1 -10804.866,E2 -10804.866} C_VEL
LIN {X 0,Y 513.78,Z 221.2,A -85,B 0,C 180,E1 -10808.28,E2 -10808.28} C_VEL
LIN {X 0,Y 513.808,Z 221.229,A -85,B 0,C 180,E1 -10811.677,E2 -10811.677} C_VEL
LIN {X 0,Y 513.812,Z 221.22,A -85,B 0,C 180,E1 -10815.231,E2 -10815.231} C_VEL
LIN {X 0,Y 513.779,Z 221.223,A -85,B 0,C 180,E1 -10818.73,E2 -10818.73} C_VEL
LIN {X 0,Y 513.779,Z 221.231,A -85,B 0,C 180,E1 -10822.303,E2 -10822.303} C_VEL
LIN {X 0,Y 513.812,Z 221.231,A -85,B 0,C 180,E1 -10825.72,E2 -10825.72} C_VEL
LIN {X 0,Y 513.801,Z 221.221,A -85,B 0,C 180,E1 -10829.24,E2 -10829.24} C_VEL
LIN {X 0,Y 513.781,Z 221.313,A -85,B 0,C 180,E1 -10832.456,E2 -10832.456} C_VEL
LIN {X 0,Y 515.013,Z 224.619,A -85,B 0,C 180,E1 -10832.93,E2 -10832.93} C_VEL
LIN {X 0,Y 516.201,Z 226.326,A -85,B 0,C 180,E1 -10833.242,E2 -10833.242} C_VEL
LIN {X 0,Y 525.585,Z 244.911,A -85,B 0,C 180,E1 -10836.047,E2 -10836.047} C_VEL
LIN {X 0,Y 535.655,Z 264.841,A -85,B 0,C 180,E1 -10838.844,E2 -10838.844} C_VEL
LIN {X 0,Y 547.492,Z 289.167,A -85,B 0,C 180,E1 -10841.946,E2 -10841.946} C_VEL
LIN {X 0,Y 554.609,Z 304.613,A -85,B 0,C 180,E1 -10843.739,E2 -10843.739} C_VEL
LIN {X 0,Y 553.588,Z 314.57,A -85,B 0,C 180,E1 -10844.321,E2 -10844.321} C_VEL
LIN {X 0,Y 556.414,Z 341.608,A -85,B 0,C 180,E1 -10845.062,E2 -10845.062} C_VEL
LIN {X 0,Y 547.903,Z 580.869,A -85,B 0,C 180,E1 -10848.765,E2 -10848.765} C_VEL
LIN {X 0,Y 544.443,Z 692.816,A -85,B 0,C 180,E1 -10850.464,E2 -10850.464} C_VEL
LIN {X 0,Y 542.93,Z 717.515,A -85,B 0,C 180,E1 -10851.016,E2 -10851.016} C_VEL
LIN {X 0,Y 541.124,Z 741.364,A -85,B 0,C 180,E1 -10851.722,E2 -10851.722} C_VEL
LIN {X 0,Y 538.988,Z 763.83,A -85,B 0,C 180,E1 -10852.581,E2 -10852.581} C_VEL
LIN {X 0,Y 536.611,Z 786.263,A -85,B 0,C 180,E1 -10853.607,E2 -10853.607} C_VEL
LIN {X 0,Y 533.939,Z 808.357,A -85,B 0,C 180,E1 -10854.841,E2 -10854.841} C_VEL
LIN {X 0,Y 531.121,Z 830.193,A -85,B 0,C 180,E1 -10856.264,E2 -10856.264} C_VEL
LIN {X 0,Y 528.363,Z 850.31,A -85,B 0,C 180,E1 -10857.809,E2 -10857.809} C_VEL
LIN {X 0,Y 525.519,Z 870.526,A -85,B 0,C 180,E1 -10859.595,E2 -10859.595} C_VEL
LIN {X 0,Y 523.04,Z 887.566,A -85,B 0,C 180,E1 -10861.339,E2 -10861.339} C_VEL
LIN {X 0,Y 520.548,Z 905.348,A -85,B 0,C 180,E1 -10863.413,E2 -10863.413} C_VEL
LIN {X 0,Y 518.526,Z 920.04,A -85,B 0,C 180,E1 -10865.385,E2 -10865.385} C_VEL
LIN {X 0,Y 516.62,Z 935.081,A -85,B 0,C 180,E1 -10867.691,E2 -10867.691} C_VEL
LIN {X 0,Y 515.125,Z 947.805,A -85,B 0,C 180,E1 -10869.964,E2 -10869.964} C_VEL
LIN {X 0,Y 513.93,Z 959.862,A -85,B 0,C 180,E1 -10872.448,E2 -10872.448} C_VEL
LIN {X 0,Y 513.116,Z 969.651,A -85,B 0,C 180,E1 -10874.863,E2 -10874.863} C_VEL
LIN {X 0,Y 512.574,Z 978.291,A -85,B 0,C 180,E1 -10877.38,E2 -10877.38} C_VEL
LIN {X 0,Y 512.276,Z 985.347,A -85,B 0,C 180,E1 -10879.996,E2 -10879.996} C_VEL
LIN {X 0,Y 512.135,Z 990.375,A -85,B 0,C 180,E1 -10882.371,E2 -10882.371} C_VEL
LIN {X 0,Y 512.127,Z 994.251,A -85,B 0,C 180,E1 -10884.96,E2 -10884.96} C_VEL
LIN {X 0,Y 512.146,Z 996.271,A -85,B 0,C 180,E1 -10887.202,E2 -10887.202} C_VEL
LIN {X 0,Y 512.166,Z 997.098,A -85,B 0,C 180,E1 -10889.329,E2 -10889.329} C_VEL
LIN {X 0,Y 512.187,Z 996.701,A -85,B 0,C 180,E1 -10891.902,E2 -10891.902} C_VEL
LIN {X 0,Y 512.182,Z 994.664,A -85,B 0,C 180,E1 -10894.367,E2 -10894.367} C_VEL
LIN {X 0,Y 512.19,Z 991.585,A -85,B 0,C 180,E1 -10896.614,E2 -10896.614} C_VEL
LIN {X 0,Y 512.276,Z 986.225,A -85,B 0,C 180,E1 -10899.323,E2 -10899.323} C_VEL
LIN {X 0,Y 512.482,Z 979.874,A -85,B 0,C 180,E1 -10901.707,E2 -10901.707} C_VEL
LIN {X 0,Y 512.885,Z 972.073,A -85,B 0,C 180,E1 -10904.105,E2 -10904.105} C_VEL
LIN {X 0,Y 513.582,Z 961.984,A -85,B 0,C 180,E1 -10906.63,E2 -10906.63} C_VEL
LIN {X 0,Y 514.442,Z 951.733,A -85,B 0,C 180,E1 -10908.823,E2 -10908.823} C_VEL
LIN {X 0,Y 515.831,Z 937.766,A -85,B 0,C 180,E1 -10911.372,E2 -10911.372} C_VEL
LIN {X 0,Y 517.342,Z 924.51,A -85,B 0,C 180,E1 -10913.462,E2 -10913.462} C_VEL
LIN {X 0,Y 519.377,Z 907.516,A -85,B 0,C 180,E1 -10915.791,E2 -10915.791} C_VEL
LIN {X 0,Y 521.504,Z 890.928,A -85,B 0,C 180,E1 -10917.769,E2 -10917.769} C_VEL
LIN {X 0,Y 523.962,Z 871.83,A -85,B 0,C 180,E1 -10919.747,E2 -10919.747} C_VEL
LIN {X 0,Y 526.505,Z 852.51,A -85,B 0,C 180,E1 -10921.493,E2 -10921.493} C_VEL
LIN {X 0,Y 529.134,Z 831.779,A -85,B 0,C 180,E1 -10923.101,E2 -10923.101} C_VEL
LIN {X 0,Y 531.627,Z 811.405,A -85,B 0,C 180,E1 -10924.481,E2 -10924.481} C_VEL
LIN {X 0,Y 534.108,Z 789.39,A -85,B 0,C 180,E1 -10925.739,E2 -10925.739} C_VEL
LIN {X 0,Y 536.515,Z 766.93,A -85,B 0,C 180,E1 -10926.828,E2 -10926.828} C_VEL
LIN {X 0,Y 538.617,Z 743.789,A -85,B 0,C 180,E1 -10927.737,E2 -10927.737} C_VEL
LIN {X 0,Y 540.513,Z 719.52,A -85,B 0,C 180,E1 -10928.498,E2 -10928.498} C_VEL
LIN {X 0,Y 541.892,Z 696.774,A -85,B 0,C 180,E1 -10929.034,E2 -10929.034} C_VEL
LIN {X 0,Y 543.2,Z 661.353,A -85,B 0,C 180,E1 -10929.614,E2 -10929.614} C_VEL
LIN {X 0,Y 546.299,Z 571.031,A -85,B 0,C 180,E1 -10931.037,E2 -10931.037} C_VEL
LIN {X 0,Y 550.506,Z 486.216,A -85,B 0,C 180,E1 -10932.524,E2 -10932.524} C_VEL
LIN {X 0,Y 555.962,Z 408.499,A -85,B 0,C 180,E1 -10934.007,E2 -10934.007} C_VEL
LIN {X 0,Y 561.718,Z 346.62,A -85,B 0,C 180,E1 -10935.273,E2 -10935.273} C_VEL
LIN {X 0,Y 563.414,Z 343.383,A -85,B 0,C 180,E1 -10935.442,E2 -10935.442} C_VEL
LIN {X 0,Y 571.56,Z 326.361,A -85,B 0,C 180,E1 -10936.992,E2 -10936.992} C_VEL
LIN {X 0,Y 573.618,Z 322.708,A -85,B 0,C 180,E1 -10937.358,E2 -10937.358} C_VEL
LIN {X 0,Y 573.653,Z 321.761,A -85,B 0,C 180,E1 -10938.253,E2 -10938.253} C_VEL
LIN {X 0,Y 573.256,Z 322.397,A -85,B 0,C 180,E1 -10938.851,E2 -10938.851} C_VEL
LIN {X 0,Y 564.185,Z 338.196,A -85,B 0,C 180,E1 -10940.598,E2 -10940.598} C_VEL
LIN {X 0,Y 555.357,Z 358.916,A -85,B 0,C 180,E1 -10942.731,E2 -10942.731} C_VEL
LIN {X 0,Y 548.201,Z 381.824,A -85,B 0,C 180,E1 -10944.932,E2 -10944.932} C_VEL
LIN {X 0,Y 545.95,Z 391.32,A -85,B 0,C 180,E1 -10945.78,E2 -10945.78} C_VEL
LIN {X 0,Y 546.136,Z 415.633,A -85,B 0,C 180,E1 -10947.327,E2 -10947.327} C_VEL
LIN {X 0,Y 546.636,Z 442.357,A -85,B 0,C 180,E1 -10948.771,E2 -10948.771} C_VEL
LIN {X 0,Y 547.093,Z 470.384,A -85,B 0,C 180,E1 -10950.085,E2 -10950.085} C_VEL
LIN {X 0,Y 547.38,Z 503.169,A -85,B 0,C 180,E1 -10951.414,E2 -10951.414} C_VEL
LIN {X 0,Y 536.921,Z 611.379,A -85,B 0,C 180,E1 -10954.036,E2 -10954.036} C_VEL
LIN {X 0,Y 530.828,Z 691.444,A -85,B 0,C 180,E1 -10955.973,E2 -10955.973} C_VEL
LIN {X 0,Y 529.01,Z 714.174,A -85,B 0,C 180,E1 -10956.732,E2 -10956.732} C_VEL
LIN {X 0,Y 527.139,Z 736.948,A -85,B 0,C 180,E1 -10957.706,E2 -10957.706} C_VEL
LIN {X 0,Y 525.344,Z 757.403,A -85,B 0,C 180,E1 -10958.8,E2 -10958.8} C_VEL
LIN {X 0,Y 523.665,Z 776.116,A -85,B 0,C 180,E1 -10960.014,E2 -10960.014} C_VEL
LIN {X 0,Y 521.997,Z 793.772,A -85,B 0,C 180,E1 -10961.402,E2 -10961.402} C_VEL
LIN {X 0,Y 520.492,Z 809.246,A -85,B 0,C 180,E1 -10962.85,E2 -10962.85} C_VEL
LIN {X 0,Y 519.102,Z 822.948,A -85,B 0,C 180,E1 -10964.386,E2 -10964.386} C_VEL
LIN {X 0,Y 517.844,Z 835.239,A -85,B 0,C 180,E1 -10966.033,E2 -10966.033} C_VEL
LIN {X 0,Y 516.683,Z 846.153,A -85,B 0,C 180,E1 -10967.823,E2 -10967.823} C_VEL
LIN {X 0,Y 515.749,Z 855.031,A -85,B 0,C 180,E1 -10969.613,E2 -10969.613} C_VEL
LIN {X 0,Y 514.958,Z 862.392,A -85,B 0,C 180,E1 -10971.514,E2 -10971.514} C_VEL
LIN {X 0,Y 514.341,Z 868.175,A -85,B 0,C 180,E1 -10973.526,E2 -10973.526} C_VEL
LIN {X 0,Y 513.885,Z 872.044,A -85,B 0,C 180,E1 -10975.536,E2 -10975.536} C_VEL
LIN {X 0,Y 513.568,Z 874.096,A -85,B 0,C 180,E1 -10977.545,E2 -10977.545} C_VEL
LIN {X 0,Y 513.371,Z 874.395,A -85,B 0,C 180,E1 -10979.554,E2 -10979.554} C_VEL
LIN {X 0,Y 513.263,Z 872.984,A -85,B 0,C 180,E1 -10981.563,E2 -10981.563} C_VEL
LIN {X 0,Y 513.257,Z 869.868,A -85,B 0,C 180,E1 -10983.574,E2 -10983.574} C_VEL
LIN {X 0,Y 513.365,Z 865.003,A -85,B 0,C 180,E1 -10985.589,E2 -10985.589} C_VEL
LIN {X 0,Y 513.607,Z 858.286,A -85,B 0,C 180,E1 -10987.607,E2 -10987.607} C_VEL
LIN {X 0,Y 514.03,Z 849.547,A -85,B 0,C 180,E1 -10989.63,E2 -10989.63} C_VEL
LIN {X 0,Y 514.645,Z 839.211,A -85,B 0,C 180,E1 -10991.544,E2 -10991.544} C_VEL
LIN {X 0,Y 515.438,Z 827.346,A -85,B 0,C 180,E1 -10993.347,E2 -10993.347} C_VEL
LIN {X 0,Y 516.435,Z 813.483,A -85,B 0,C 180,E1 -10995.095,E2 -10995.095} C_VEL
LIN {X 0,Y 517.549,Z 798.451,A -85,B 0,C 180,E1 -10996.672,E2 -10996.672} C_VEL
LIN {X 0,Y 518.745,Z 782.464,A -85,B 0,C 180,E1 -10998.079,E2 -10998.079} C_VEL
LIN {X 0,Y 519.999,Z 764.842,A -85,B 0,C 180,E1 -10999.372,E2 -10999.372} C_VEL
LIN {X 0,Y 521.266,Z 746.492,A -85,B 0,C 180,E1 -11000.479,E2 -11000.479} C_VEL
LIN {X 0,Y 522.517,Z 726.749,A -85,B 0,C 180,E1 -11001.438,E2 -11001.438} C_VEL
LIN {X 0,Y 523.668,Z 705.694,A -85,B 0,C 180,E1 -11002.232,E2 -11002.232} C_VEL
LIN {X 0,Y 524.648,Z 684.535,A -85,B 0,C 180,E1 -11002.813,E2 -11002.813} C_VEL
LIN {X 0,Y 526.783,Z 615.83,A -85,B 0,C 180,E1 -11004.044,E2 -11004.044} C_VEL
LIN {X 0,Y 530.822,Z 495.843,A -85,B 0,C 180,E1 -11006.166,E2 -11006.166} C_VEL
LIN {X 0,Y 526.163,Z 448.839,A -85,B 0,C 180,E1 -11007.38,E2 -11007.38} C_VEL
LIN {X 0,Y 530.122,Z 393.926,A -85,B 0,C 180,E1 -11011.245,E2 -11011.245} C_VEL
LIN {X 0,Y 533.885,Z 347.053,A -85,B 0,C 180,E1 -11014.575,E2 -11014.575} C_VEL
LIN {X 0,Y 538.606,Z 293.929,A -85,B 0,C 180,E1 -11018.388,E2 -11018.388} C_VEL
LIN {X 0,Y 539.286,Z 285.255,A -85,B 0,C 180,E1 -11019.025,E2 -11019.025} C_VEL
LIN {X 0,Y 530.654,Z 262.108,A -85,B 0,C 180,E1 -11021.578,E2 -11021.578} C_VEL
LIN {X 0,Y 524.046,Z 245.633,A -85,B 0,C 180,E1 -11023.535,E2 -11023.535} C_VEL
LIN {X 0,Y 525.887,Z 246.35,A -85,B 0,C 180,E1 -11023.796,E2 -11023.796} C_VEL
LIN {X 0,Y 526.934,Z 246.319,A -85,B 0,C 180,E1 -11023.913,E2 -11023.913} C_VEL
LIN {X 0,Y 535.312,Z 264.189,A -85,B 0,C 180,E1 -11026.137,E2 -11026.137} C_VEL
LIN {X 0,Y 543.501,Z 284.174,A -85,B 0,C 180,E1 -11028.484,E2 -11028.484} C_VEL
LIN {X 0,Y 548.692,Z 298.744,A -85,B 0,C 180,E1 -11030.103,E2 -11030.103} C_VEL
LIN {X 0,Y 548.114,Z 340.328,A -85,B 0,C 180,E1 -11032.987,E2 -11032.987} C_VEL
LIN {X 0,Y 548.17,Z 350.473,A -85,B 0,C 180,E1 -11033.643,E2 -11033.643} C_VEL
LIN {X 0,Y 547.836,Z 351.92,A -85,B 0,C 180,E1 -11033.701,E2 -11033.701} C_VEL
LIN {X 0,Y 545.728,Z 359.167,A -85,B 0,C 180,E1 -11033.883,E2 -11033.883} C_VEL
LIN {X 0,Y 541.701,Z 370.787,A -85,B 0,C 180,E1 -11033.906,E2 -11033.906} C_VEL
LIN {X 0,Y 539.162,Z 380.551,A -85,B 0,C 180,E1 -11033.881,E2 -11033.881} C_VEL
LIN {X 0,Y 538.574,Z 386.081,A -85,B 0,C 180,E1 -11033.926,E2 -11033.926} C_VEL
LIN {X 0,Y 536.112,Z 460.229,A -85,B 0,C 180,E1 -11035.047,E2 -11035.047} C_VEL
LIN {X 0,Y 532.615,Z 535.506,A -85,B 0,C 180,E1 -11036.375,E2 -11036.375} C_VEL
LIN {X 0,Y 527.969,Z 619.963,A -85,B 0,C 180,E1 -11038.08,E2 -11038.08} C_VEL
LIN {X 0,Y 526.652,Z 649.813,A -85,B 0,C 180,E1 -11038.805,E2 -11038.805} C_VEL
LIN {X 0,Y 525.398,Z 671.372,A -85,B 0,C 180,E1 -11039.524,E2 -11039.524} C_VEL
LIN {X 0,Y 523.721,Z 693.609,A -85,B 0,C 180,E1 -11040.49,E2 -11040.49} C_VEL
LIN {X 0,Y 521.795,Z 714.5,A -85,B 0,C 180,E1 -11041.626,E2 -11041.626} C_VEL
LIN {X 0,Y 519.775,Z 733.497,A -85,B 0,C 180,E1 -11042.876,E2 -11042.876} C_VEL
LIN {X 0,Y 517.656,Z 751.757,A -85,B 0,C 180,E1 -11044.301,E2 -11044.301} C_VEL
LIN {X 0,Y 515.416,Z 769.759,A -85,B 0,C 180,E1 -11045.959,E2 -11045.959} C_VEL
LIN {X 0,Y 513.35,Z 785.828,A -85,B 0,C 180,E1 -11047.698,E2 -11047.698} C_VEL
LIN {X 0,Y 511.482,Z 800.258,A -85,B 0,C 180,E1 -11049.517,E2 -11049.517} C_VEL
LIN {X 0,Y 509.605,Z 814.92,A -85,B 0,C 180,E1 -11051.703,E2 -11051.703} C_VEL
LIN {X 0,Y 508.104,Z 827.192,A -85,B 0,C 180,E1 -11053.891,E2 -11053.891} C_VEL
LIN {X 0,Y 506.952,Z 837.449,A -85,B 0,C 180,E1 -11056.076,E2 -11056.076} C_VEL
LIN {X 0,Y 506.087,Z 846.355,A -85,B 0,C 180,E1 -11058.374,E2 -11058.374} C_VEL
LIN {X 0,Y 505.478,Z 853.506,A -85,B 0,C 180,E1 -11060.665,E2 -11060.665} C_VEL
LIN {X 0,Y 505.1,Z 859.21,A -85,B 0,C 180,E1 -11063.064,E2 -11063.064} C_VEL
LIN {X 0,Y 504.891,Z 863.141,A -85,B 0,C 180,E1 -11065.456,E2 -11065.456} C_VEL
LIN {X 0,Y 504.788,Z 865.457,A -85,B 0,C 180,E1 -11067.843,E2 -11067.843} C_VEL
LIN {X 0,Y 504.765,Z 866.186,A -85,B 0,C 180,E1 -11070.227,E2 -11070.227} C_VEL
LIN {X 0,Y 504.792,Z 865.243,A -85,B 0,C 180,E1 -11072.611,E2 -11072.611} C_VEL
LIN {X 0,Y 504.912,Z 862.638,A -85,B 0,C 180,E1 -11074.999,E2 -11074.999} C_VEL
LIN {X 0,Y 505.142,Z 858.169,A -85,B 0,C 180,E1 -11077.507,E2 -11077.507} C_VEL
LIN {X 0,Y 505.561,Z 852.489,A -85,B 0,C 180,E1 -11079.793,E2 -11079.793} C_VEL
LIN {X 0,Y 506.247,Z 844.704,A -85,B 0,C 180,E1 -11082.201,E2 -11082.201} C_VEL
LIN {X 0,Y 507.204,Z 835.165,A -85,B 0,C 180,E1 -11084.545,E2 -11084.545} C_VEL
LIN {X 0,Y 508.42,Z 824.501,A -85,B 0,C 180,E1 -11086.71,E2 -11086.71} C_VEL
LIN {X 0,Y 509.982,Z 811.826,A -85,B 0,C 180,E1 -11088.875,E2 -11088.875} C_VEL
LIN {X 0,Y 511.731,Z 798.33,A -85,B 0,C 180,E1 -11090.831,E2 -11090.831} C_VEL
LIN {X 0,Y 513.696,Z 783.374,A -85,B 0,C 180,E1 -11092.687,E2 -11092.687} C_VEL
LIN {X 0,Y 515.928,Z 766.106,A -85,B 0,C 180,E1 -11094.503,E2 -11094.503} C_VEL
LIN {X 0,Y 518.212,Z 747.418,A -85,B 0,C 180,E1 -11096.161,E2 -11096.161} C_VEL
LIN {X 0,Y 520.39,Z 728.283,A -85,B 0,C 180,E1 -11097.585,E2 -11097.585} C_VEL
LIN {X 0,Y 522.309,Z 709.125,A -85,B 0,C 180,E1 -11098.781,E2 -11098.781} C_VEL
LIN {X 0,Y 524.169,Z 688.135,A -85,B 0,C 180,E1 -11099.86,E2 -11099.86} C_VEL
LIN {X 0,Y 525.754,Z 666.086,A -85,B 0,C 180,E1 -11100.761,E2 -11100.761} C_VEL
LIN {X 0,Y 526.902,Z 644.598,A -85,B 0,C 180,E1 -11101.436,E2 -11101.436} C_VEL
LIN {X 0,Y 528.98,Z 602.126,A -85,B 0,C 180,E1 -11102.395,E2 -11102.395} C_VEL
LIN {X 0,Y 533.44,Z 520.097,A -85,B 0,C 180,E1 -11104.006,E2 -11104.006} C_VEL
LIN {X 0,Y 536.587,Z 449.175,A -85,B 0,C 180,E1 -11105.225,E2 -11105.225} C_VEL
LIN {X 0,Y 539.419,Z 363.626,A -85,B 0,C 180,E1 -11106.514,E2 -11106.514} C_VEL
LIN {X 0,Y 542.032,Z 351.759,A -85,B 0,C 180,E1 -11106.988,E2 -11106.988} C_VEL
LIN {X 0,Y 542.205,Z 315.561,A -85,B 0,C 180,E1 -11109.435,E2 -11109.435} C_VEL
LIN {X 0,Y 542.378,Z 301.936,A -85,B 0,C 180,E1 -11110.414,E2 -11110.414} C_VEL
LIN {X 0,Y 535.091,Z 282.309,A -85,B 0,C 180,E1 -11112.666,E2 -11112.666} C_VEL
LIN {X 0,Y 527.023,Z 263.385,A -85,B 0,C 180,E1 -11114.954,E2 -11114.954} C_VEL
LIN {X 0,Y 518.207,Z 245.125,A -85,B 0,C 180,E1 -11117.295,E2 -11117.295} C_VEL
LIN {X 0,Y 510.724,Z 231.488,A -85,B 0,C 180,E1 -11119.163,E2 -11119.163} C_VEL
LIN {X 0,Y 508.165,Z 226.883,A -85,B 0,C 180,E1 -11119.805,E2 -11119.805} C_VEL
LIN {X 0,Y 506.179,Z 223.633,A -85,B 0,C 180,E1 -11120.28,E2 -11120.28} C_VEL
LIN {X 0,Y 505.871,Z 222.206,A -85,B 0,C 180,E1 -11120.431,E2 -11120.431} C_VEL
LIN {X 0,Y 505.864,Z 222.201,A -85,B 0,C 180,E1 -11123.943,E2 -11123.943} C_VEL
LIN {X 0,Y 505.859,Z 222.193,A -85,B 0,C 180,E1 -11127.477,E2 -11127.477} C_VEL
LIN {X 0,Y 505.857,Z 222.193,A -85,B 0,C 180,E1 -11131.035,E2 -11131.035} C_VEL
LIN {X 0,Y 505.868,Z 222.213,A -85,B 0,C 180,E1 -11134.601,E2 -11134.601} C_VEL
LIN {X 0,Y 505.859,Z 222.205,A -85,B 0,C 180,E1 -11138.185,E2 -11138.185} C_VEL
LIN {X 0,Y 505.862,Z 222.18,A -85,B 0,C 180,E1 -11141.683,E2 -11141.683} C_VEL
LIN {X 0,Y 505.864,Z 222.215,A -85,B 0,C 180,E1 -11145.227,E2 -11145.227} C_VEL
LIN {X 0,Y 505.858,Z 222.186,A -85,B 0,C 180,E1 -11148.715,E2 -11148.715} C_VEL
LIN {X 0,Y 505.851,Z 222.204,A -85,B 0,C 180,E1 -11152.275,E2 -11152.275} C_VEL
LIN {X 0,Y 505.861,Z 222.199,A -85,B 0,C 180,E1 -11155.806,E2 -11155.806} C_VEL
LIN {X 0,Y 505.864,Z 222.188,A -85,B 0,C 180,E1 -11159.32,E2 -11159.32} C_VEL
LIN {X 0,Y 505.855,Z 222.213,A -85,B 0,C 180,E1 -11162.832,E2 -11162.832} C_VEL
LIN {X 0,Y 505.84,Z 222.182,A -85,B 0,C 180,E1 -11166.355,E2 -11166.355} C_VEL
LIN {X 0,Y 505.862,Z 222.216,A -85,B 0,C 180,E1 -11169.902,E2 -11169.902} C_VEL
LIN {X 0,Y 505.872,Z 222.216,A -85,B 0,C 180,E1 -11173.488,E2 -11173.488} C_VEL
LIN {X 0,Y 505.85,Z 222.219,A -85,B 0,C 180,E1 -11176.922,E2 -11176.922} C_VEL
LIN {X 0,Y 505.837,Z 222.219,A -85,B 0,C 180,E1 -11180.48,E2 -11180.48} C_VEL
LIN {X 0,Y 505.863,Z 222.211,A -85,B 0,C 180,E1 -11183.904,E2 -11183.904} C_VEL
LIN {X 0,Y 505.873,Z 222.21,A -85,B 0,C 180,E1 -11187.442,E2 -11187.442} C_VEL
LIN {X 0,Y 505.833,Z 222.221,A -85,B 0,C 180,E1 -11190.795,E2 -11190.795} C_VEL
LIN {X 0,Y 505.912,Z 222.453,A -85,B 0,C 180,E1 -11191.542,E2 -11191.542} C_VEL
LIN {X 0,Y 507.3,Z 225.898,A -85,B 0,C 180,E1 -11192.056,E2 -11192.056} C_VEL
LIN {X 0,Y 508.301,Z 227.618,A -85,B 0,C 180,E1 -11192.348,E2 -11192.348} C_VEL
LIN {X 0,Y 513.311,Z 237.529,A -85,B 0,C 180,E1 -11193.92,E2 -11193.92} C_VEL
LIN {X 0,Y 521.601,Z 253.365,A -85,B 0,C 180,E1 -11196.324,E2 -11196.324} C_VEL
LIN {X 0,Y 532.956,Z 276.351,A -85,B 0,C 180,E1 -11199.495,E2 -11199.495} C_VEL
LIN {X 0,Y 544.952,Z 301.312,A -85,B 0,C 180,E1 -11202.614,E2 -11202.614} C_VEL
LIN {X 0,Y 547.961,Z 307.788,A -85,B 0,C 180,E1 -11203.367,E2 -11203.367} C_VEL
LIN {X 0,Y 547.233,Z 315.374,A -85,B 0,C 180,E1 -11203.808,E2 -11203.808} C_VEL
LIN {X 0,Y 550.059,Z 342.901,A -85,B 0,C 180,E1 -11204.569,E2 -11204.569} C_VEL
LIN {X 0,Y 541.407,Z 573.916,A -85,B 0,C 180,E1 -11208.201,E2 -11208.201} C_VEL
LIN {X 0,Y 537.523,Z 692.937,A -85,B 0,C 180,E1 -11210.038,E2 -11210.038} C_VEL
LIN {X 0,Y 535.962,Z 717.382,A -85,B 0,C 180,E1 -11210.593,E2 -11210.593} C_VEL
LIN {X 0,Y 534.114,Z 740.937,A -85,B 0,C 180,E1 -11211.298,E2 -11211.298} C_VEL
LIN {X 0,Y 531.911,Z 763.372,A -85,B 0,C 180,E1 -11212.164,E2 -11212.164} C_VEL
LIN {X 0,Y 529.409,Z 786.177,A -85,B 0,C 180,E1 -11213.222,E2 -11213.222} C_VEL
LIN {X 0,Y 526.634,Z 808.439,A -85,B 0,C 180,E1 -11214.48,E2 -11214.48} C_VEL
LIN {X 0,Y 523.723,Z 830.244,A -85,B 0,C 180,E1 -11215.92,E2 -11215.92} C_VEL
LIN {X 0,Y 521.006,Z 849.376,A -85,B 0,C 180,E1 -11217.406,E2 -11217.406} C_VEL
LIN {X 0,Y 518.114,Z 869.305,A -85,B 0,C 180,E1 -11219.182,E2 -11219.182} C_VEL
LIN {X 0,Y 515.412,Z 887.271,A -85,B 0,C 180,E1 -11221.037,E2 -11221.037} C_VEL
LIN {X 0,Y 512.864,Z 904.788,A -85,B 0,C 180,E1 -11223.108,E2 -11223.108} C_VEL
LIN {X 0,Y 510.766,Z 919.47,A -85,B 0,C 180,E1 -11225.109,E2 -11225.109} C_VEL
LIN {X 0,Y 508.759,Z 934.69,A -85,B 0,C 180,E1 -11227.476,E2 -11227.476} C_VEL
LIN {X 0,Y 507.261,Z 946.969,A -85,B 0,C 180,E1 -11229.701,E2 -11229.701} C_VEL
LIN {X 0,Y 506.043,Z 958.805,A -85,B 0,C 180,E1 -11232.166,E2 -11232.166} C_VEL
LIN {X 0,Y 505.181,Z 968.655,A -85,B 0,C 180,E1 -11234.62,E2 -11234.62} C_VEL
LIN {X 0,Y 504.625,Z 977.193,A -85,B 0,C 180,E1 -11237.13,E2 -11237.13} C_VEL
LIN {X 0,Y 504.311,Z 984.173,A -85,B 0,C 180,E1 -11239.721,E2 -11239.721} C_VEL
LIN {X 0,Y 504.188,Z 989.053,A -85,B 0,C 180,E1 -11242.02,E2 -11242.02} C_VEL
LIN {X 0,Y 504.155,Z 993.143,A -85,B 0,C 180,E1 -11244.651,E2 -11244.651} C_VEL
LIN {X 0,Y 504.189,Z 995.338,A -85,B 0,C 180,E1 -11247.044,E2 -11247.044} C_VEL
LIN {X 0,Y 504.215,Z 996.212,A -85,B 0,C 180,E1 -11249.205,E2 -11249.205} C_VEL
LIN {X 0,Y 504.234,Z 995.94,A -85,B 0,C 180,E1 -11251.591,E2 -11251.591} C_VEL
LIN {X 0,Y 504.225,Z 994.014,A -85,B 0,C 180,E1 -11254.208,E2 -11254.208} C_VEL
LIN {X 0,Y 504.228,Z 990.823,A -85,B 0,C 180,E1 -11256.605,E2 -11256.605} C_VEL
LIN {X 0,Y 504.291,Z 985.794,A -85,B 0,C 180,E1 -11259.242,E2 -11259.242} C_VEL
LIN {X 0,Y 504.507,Z 979.183,A -85,B 0,C 180,E1 -11261.779,E2 -11261.779} C_VEL
LIN {X 0,Y 504.889,Z 971.777,A -85,B 0,C 180,E1 -11264.099,E2 -11264.099} C_VEL
LIN {X 0,Y 505.631,Z 961.351,A -85,B 0,C 180,E1 -11266.781,E2 -11266.781} C_VEL
LIN {X 0,Y 506.522,Z 951.105,A -85,B 0,C 180,E1 -11269.009,E2 -11269.009} C_VEL
LIN {X 0,Y 507.96,Z 937.185,A -85,B 0,C 180,E1 -11271.599,E2 -11271.599} C_VEL
LIN {X 0,Y 509.531,Z 923.967,A -85,B 0,C 180,E1 -11273.721,E2 -11273.721} C_VEL
LIN {X 0,Y 511.665,Z 907.04,A -85,B 0,C 180,E1 -11276.084,E2 -11276.084} C_VEL
LIN {X 0,Y 513.877,Z 890.498,A -85,B 0,C 180,E1 -11278.091,E2 -11278.091} C_VEL
LIN {X 0,Y 516.545,Z 870.902,A -85,B 0,C 180,E1 -11280.154,E2 -11280.154} C_VEL
LIN {X 0,Y 519.296,Z 851.043,A -85,B 0,C 180,E1 -11281.972,E2 -11281.972} C_VEL
LIN {X 0,Y 522.059,Z 830.12,A -85,B 0,C 180,E1 -11283.609,E2 -11283.609} C_VEL
LIN {X 0,Y 524.827,Z 808.73,A -85,B 0,C 180,E1 -11285.059,E2 -11285.059} C_VEL
LIN {X 0,Y 527.212,Z 788.677,A -85,B 0,C 180,E1 -11286.212,E2 -11286.212} C_VEL
LIN {X 0,Y 529.764,Z 766.004,A -85,B 0,C 180,E1 -11287.325,E2 -11287.325} C_VEL
LIN {X 0,Y 531.957,Z 743.277,A -85,B 0,C 180,E1 -11288.231,E2 -11288.231} C_VEL
LIN {X 0,Y 533.987,Z 718.66,A -85,B 0,C 180,E1 -11289.014,E2 -11289.014} C_VEL
LIN {X 0,Y 535.478,Z 695.689,A -85,B 0,C 180,E1 -11289.561,E2 -11289.561} C_VEL
LIN {X 0,Y 536.94,Z 659.167,A -85,B 0,C 180,E1 -11290.169,E2 -11290.169} C_VEL
LIN {X 0,Y 540.255,Z 574.178,A -85,B 0,C 180,E1 -11291.557,E2 -11291.557} C_VEL
LIN {X 0,Y 544.753,Z 493.17,A -85,B 0,C 180,E1 -11293.023,E2 -11293.023} C_VEL
LIN {X 0,Y 550.596,Z 417.849,A -85,B 0,C 180,E1 -11294.506,E2 -11294.506} C_VEL
LIN {X 0,Y 557.665,Z 349.724,A -85,B 0,C 180,E1 -11295.94,E2 -11295.94} C_VEL
LIN {X 0,Y 559.722,Z 346.061,A -85,B 0,C 180,E1 -11296.122,E2 -11296.122} C_VEL
LIN {X 0,Y 568.341,Z 329.893,A -85,B 0,C 180,E1 -11297.639,E2 -11297.639} C_VEL
LIN {X 0,Y 569.005,Z 328.713,A -85,B 0,C 180,E1 -11297.79,E2 -11297.79} C_VEL
LIN {X 0,Y 569.057,Z 328.367,A -85,B 0,C 180,E1 -11298.245,E2 -11298.245} C_VEL
LIN {X 0,Y 568.745,Z 328.729,A -85,B 0,C 180,E1 -11298.487,E2 -11298.487} C_VEL
LIN {X 0,Y 558.919,Z 344.974,A -85,B 0,C 180,E1 -11300.308,E2 -11300.308} C_VEL
LIN {X 0,Y 550.447,Z 363.444,A -85,B 0,C 180,E1 -11302.254,E2 -11302.254} C_VEL
LIN {X 0,Y 543.053,Z 385.211,A -85,B 0,C 180,E1 -11304.396,E2 -11304.396} C_VEL
LIN {X 0,Y 542.395,Z 404.872,A -85,B 0,C 180,E1 -11305.788,E2 -11305.788} C_VEL
LIN {X 0,Y 542.184,Z 427.764,A -85,B 0,C 180,E1 -11307.195,E2 -11307.195} C_VEL
LIN {X 0,Y 542.214,Z 456.835,A -85,B 0,C 180,E1 -11308.727,E2 -11308.727} C_VEL
LIN {X 0,Y 542.175,Z 489.262,A -85,B 0,C 180,E1 -11310.182,E2 -11310.182} C_VEL
LIN {X 0,Y 541.913,Z 505.914,A -85,B 0,C 180,E1 -11310.832,E2 -11310.832} C_VEL
LIN {X 0,Y 530.594,Z 615.774,A -85,B 0,C 180,E1 -11313.563,E2 -11313.563} C_VEL
LIN {X 0,Y 524.44,Z 690.806,A -85,B 0,C 180,E1 -11315.434,E2 -11315.434} C_VEL
LIN {X 0,Y 522.323,Z 715.201,A -85,B 0,C 180,E1 -11316.266,E2 -11316.266} C_VEL
LIN {X 0,Y 520.379,Z 737.047,A -85,B 0,C 180,E1 -11317.221,E2 -11317.221} C_VEL
LIN {X 0,Y 518.289,Z 759.221,A -85,B 0,C 180,E1 -11318.431,E2 -11318.431} C_VEL
LIN {X 0,Y 516.488,Z 777.69,A -85,B 0,C 180,E1 -11319.665,E2 -11319.665} C_VEL
LIN {X 0,Y 514.728,Z 795.255,A -85,B 0,C 180,E1 -11321.07,E2 -11321.07} C_VEL
LIN {X 0,Y 513.112,Z 810.559,A -85,B 0,C 180,E1 -11322.537,E2 -11322.537} C_VEL
LIN {X 0,Y 511.616,Z 824.465,A -85,B 0,C 180,E1 -11324.121,E2 -11324.121} C_VEL
LIN {X 0,Y 510.238,Z 836.828,A -85,B 0,C 180,E1 -11325.821,E2 -11325.821} C_VEL
LIN {X 0,Y 509.089,Z 847.114,A -85,B 0,C 180,E1 -11327.523,E2 -11327.523} C_VEL
LIN {X 0,Y 508.004,Z 856.463,A -85,B 0,C 180,E1 -11329.453,E2 -11329.453} C_VEL
LIN {X 0,Y 507.164,Z 863.792,A -85,B 0,C 180,E1 -11331.383,E2 -11331.383} C_VEL
LIN {X 0,Y 506.496,Z 869.496,A -85,B 0,C 180,E1 -11333.425,E2 -11333.425} C_VEL
LIN {X 0,Y 506.002,Z 873.287,A -85,B 0,C 180,E1 -11335.466,E2 -11335.466} C_VEL
LIN {X 0,Y 505.66,Z 875.269,A -85,B 0,C 180,E1 -11337.507,E2 -11337.507} C_VEL
LIN {X 0,Y 505.448,Z 875.491,A -85,B 0,C 180,E1 -11339.547,E2 -11339.547} C_VEL
LIN {X 0,Y 505.328,Z 873.985,A -85,B 0,C 180,E1 -11341.587,E2 -11341.587} C_VEL
LIN {X 0,Y 505.318,Z 870.766,A -85,B 0,C 180,E1 -11343.63,E2 -11343.63} C_VEL
LIN {X 0,Y 505.433,Z 865.768,A -85,B 0,C 180,E1 -11345.686,E2 -11345.686} C_VEL
LIN {X 0,Y 505.686,Z 858.959,A -85,B 0,C 180,E1 -11347.727,E2 -11347.727} C_VEL
LIN {X 0,Y 506.1,Z 850.635,A -85,B 0,C 180,E1 -11349.668,E2 -11349.668} C_VEL
LIN {X 0,Y 506.732,Z 840.288,A -85,B 0,C 180,E1 -11351.611,E2 -11351.611} C_VEL
LIN {X 0,Y 507.547,Z 828.415,A -85,B 0,C 180,E1 -11353.442,E2 -11353.442} C_VEL
LIN {X 0,Y 508.537,Z 815.041,A -85,B 0,C 180,E1 -11355.16,E2 -11355.16} C_VEL
LIN {X 0,Y 509.713,Z 799.72,A -85,B 0,C 180,E1 -11356.804,E2 -11356.804} C_VEL
LIN {X 0,Y 511.008,Z 782.908,A -85,B 0,C 180,E1 -11358.304,E2 -11358.304} C_VEL
LIN {X 0,Y 512.307,Z 765.224,A -85,B 0,C 180,E1 -11359.615,E2 -11359.615} C_VEL
LIN {X 0,Y 513.637,Z 746.61,A -85,B 0,C 180,E1 -11360.751,E2 -11360.751} C_VEL
LIN {X 0,Y 514.993,Z 725.822,A -85,B 0,C 180,E1 -11361.767,E2 -11361.767} C_VEL
LIN {X 0,Y 516.161,Z 705.108,A -85,B 0,C 180,E1 -11362.551,E2 -11362.551} C_VEL
LIN {X 0,Y 517.179,Z 683.961,A -85,B 0,C 180,E1 -11363.135,E2 -11363.135} C_VEL
LIN {X 0,Y 523.62,Z 496.861,A -85,B 0,C 180,E1 -11366.53,E2 -11366.53} C_VEL
LIN {X 0,Y 518.851,Z 448.174,A -85,B 0,C 180,E1 -11367.804,E2 -11367.804} C_VEL
LIN {X 0,Y 522.969,Z 393.462,A -85,B 0,C 180,E1 -11371.699,E2 -11371.699} C_VEL
LIN {X 0,Y 526.943,Z 346.207,A -85,B 0,C 180,E1 -11375.096,E2 -11375.096} C_VEL
LIN {X 0,Y 531.809,Z 293.798,A -85,B 0,C 180,E1 -11378.901,E2 -11378.901} C_VEL
LIN {X 0,Y 532.299,Z 288.48,A -85,B 0,C 180,E1 -11379.293,E2 -11379.293} C_VEL
LIN {X 0,Y 524.104,Z 266.395,A -85,B 0,C 180,E1 -11381.759,E2 -11381.759} C_VEL
LIN {X 0,Y 518.678,Z 252.705,A -85,B 0,C 180,E1 -11383.413,E2 -11383.413} C_VEL
LIN {X 0,Y 520.86,Z 253.372,A -85,B 0,C 180,E1 -11383.717,E2 -11383.717} C_VEL
LIN {X 0,Y 522.469,Z 253.675,A -85,B 0,C 180,E1 -11383.928,E2 -11383.928} C_VEL
LIN {X 0,Y 530.14,Z 270.546,A -85,B 0,C 180,E1 -11386.046,E2 -11386.046} C_VEL
LIN {X 0,Y 537.771,Z 289.424,A -85,B 0,C 180,E1 -11388.269,E2 -11388.269} C_VEL
LIN {X 0,Y 542.432,Z 302.595,A -85,B 0,C 180,E1 -11389.743,E2 -11389.743} C_VEL
LIN {X 0,Y 541.888,Z 344.229,A -85,B 0,C 180,E1 -11392.622,E2 -11392.622} C_VEL
LIN {X 0,Y 541.832,Z 352.535,A -85,B 0,C 180,E1 -11393.148,E2 -11393.148} C_VEL
LIN {X 0,Y 539.175,Z 365.352,A -85,B 0,C 180,E1 -11393.628,E2 -11393.628} C_VEL
LIN {X 0,Y 538.574,Z 386.081,A -85,B 0,C 180,E1 -11393.926,E2 -11393.926} C_VEL
LIN {X 0,Y 537.549,Z 393.768,A -85,B 0,C 180,E1 -11393.972,E2 -11393.972} C_VEL
LIN {X 0,Y 531.97,Z 414.245,A -85,B 0,C 180,E1 -11393.868,E2 -11393.868} C_VEL
LIN {X 0,Y 531.147,Z 420.838,A -85,B 0,C 180,E1 -11393.918,E2 -11393.918} C_VEL
LIN {X 0,Y 528.344,Z 490.186,A -85,B 0,C 180,E1 -11395.045,E2 -11395.045} C_VEL
LIN {X 0,Y 524.295,Z 567.12,A -85,B 0,C 180,E1 -11396.496,E2 -11396.496} C_VEL
LIN {X 0,Y 520.473,Z 635.606,A -85,B 0,C 180,E1 -11397.967,E2 -11397.967} C_VEL
LIN {X 0,Y 519.366,Z 658.237,A -85,B 0,C 180,E1 -11398.596,E2 -11398.596} C_VEL
LIN {X 0,Y 517.948,Z 679.647,A -85,B 0,C 180,E1 -11399.392,E2 -11399.392} C_VEL
LIN {X 0,Y 516.172,Z 700.962,A -85,B 0,C 180,E1 -11400.398,E2 -11400.398} C_VEL
LIN {X 0,Y 514.095,Z 721.659,A -85,B 0,C 180,E1 -11401.605,E2 -11401.605} C_VEL
LIN {X 0,Y 511.877,Z 741.271,A -85,B 0,C 180,E1 -11402.989,E2 -11402.989} C_VEL
LIN {X 0,Y 509.646,Z 759.198,A -85,B 0,C 180,E1 -11404.488,E2 -11404.488} C_VEL
LIN {X 0,Y 507.324,Z 776.844,A -85,B 0,C 180,E1 -11406.231,E2 -11406.231} C_VEL
LIN {X 0,Y 505.075,Z 793.275,A -85,B 0,C 180,E1 -11408.15,E2 -11408.15} C_VEL
LIN {X 0,Y 502.998,Z 808.447,A -85,B 0,C 180,E1 -11410.249,E2 -11410.249} C_VEL
LIN {X 0,Y 501.291,Z 821.269,A -85,B 0,C 180,E1 -11412.351,E2 -11412.351} C_VEL
LIN {X 0,Y 499.859,Z 832.688,A -85,B 0,C 180,E1 -11414.571,E2 -11414.571} C_VEL
LIN {X 0,Y 498.729,Z 842.666,A -85,B 0,C 180,E1 -11416.906,E2 -11416.906} C_VEL
LIN {X 0,Y 497.931,Z 850.784,A -85,B 0,C 180,E1 -11419.237,E2 -11419.237} C_VEL
LIN {X 0,Y 497.386,Z 857.452,A -85,B 0,C 180,E1 -11421.678,E2 -11421.678} C_VEL
LIN {X 0,Y 497.063,Z 862.275,A -85,B 0,C 180,E1 -11424.111,E2 -11424.111} C_VEL
LIN {X 0,Y 496.894,Z 865.442,A -85,B 0,C 180,E1 -11426.539,E2 -11426.539} C_VEL
LIN {X 0,Y 496.823,Z 867.011,A -85,B 0,C 180,E1 -11428.962,E2 -11428.962} C_VEL
LIN {X 0,Y 496.828,Z 866.984,A -85,B 0,C 180,E1 -11431.268,E2 -11431.268} C_VEL
LIN {X 0,Y 496.892,Z 865.419,A -85,B 0,C 180,E1 -11433.576,E2 -11433.576} C_VEL
LIN {X 0,Y 497.066,Z 862.234,A -85,B 0,C 180,E1 -11436.004,E2 -11436.004} C_VEL
LIN {X 0,Y 497.391,Z 857.399,A -85,B 0,C 180,E1 -11438.439,E2 -11438.439} C_VEL
LIN {X 0,Y 497.95,Z 850.629,A -85,B 0,C 180,E1 -11440.91,E2 -11440.91} C_VEL
LIN {X 0,Y 498.743,Z 842.577,A -85,B 0,C 180,E1 -11443.212,E2 -11443.212} C_VEL
LIN {X 0,Y 499.878,Z 832.577,A -85,B 0,C 180,E1 -11445.547,E2 -11445.547} C_VEL
LIN {X 0,Y 501.315,Z 821.132,A -85,B 0,C 180,E1 -11447.768,E2 -11447.768} C_VEL
LIN {X 0,Y 503.031,Z 808.281,A -85,B 0,C 180,E1 -11449.871,E2 -11449.871} C_VEL
LIN {X 0,Y 504.99,Z 793.993,A -85,B 0,C 180,E1 -11451.854,E2 -11451.854} C_VEL
LIN {X 0,Y 507.146,Z 778.179,A -85,B 0,C 180,E1 -11453.716,E2 -11453.716} C_VEL
LIN {X 0,Y 509.359,Z 761.425,A -85,B 0,C 180,E1 -11455.399,E2 -11455.399} C_VEL
LIN {X 0,Y 511.671,Z 743.145,A -85,B 0,C 180,E1 -11456.96,E2 -11456.96} C_VEL
LIN {X 0,Y 513.878,Z 723.908,A -85,B 0,C 180,E1 -11458.344,E2 -11458.344} C_VEL
LIN {X 0,Y 515.863,Z 704.567,A -85,B 0,C 180,E1 -11459.507,E2 -11459.507} C_VEL
LIN {X 0,Y 517.689,Z 683.844,A -85,B 0,C 180,E1 -11460.529,E2 -11460.529} C_VEL
LIN {X 0,Y 519.229,Z 661.611,A -85,B 0,C 180,E1 -11461.393,E2 -11461.393} C_VEL
LIN {X 0,Y 520.365,Z 638.867,A -85,B 0,C 180,E1 -11462.05,E2 -11462.05} C_VEL
LIN {X 0,Y 523.744,Z 577.359,A -85,B 0,C 180,E1 -11463.392,E2 -11463.392} C_VEL
LIN {X 0,Y 527.915,Z 499.903,A -85,B 0,C 180,E1 -11464.877,E2 -11464.877} C_VEL
LIN {X 0,Y 530.827,Z 431.423,A -85,B 0,C 180,E1 -11466.017,E2 -11466.017} C_VEL
LIN {X 0,Y 532.847,Z 366.95,A -85,B 0,C 180,E1 -11466.972,E2 -11466.972} C_VEL
LIN {X 0,Y 535.831,Z 353.175,A -85,B 0,C 180,E1 -11467.526,E2 -11467.526} C_VEL
LIN {X 0,Y 536.059,Z 315.952,A -85,B 0,C 180,E1 -11470.054,E2 -11470.054} C_VEL
LIN {X 0,Y 536.161,Z 305.817,A -85,B 0,C 180,E1 -11470.786,E2 -11470.786} C_VEL
LIN {X 0,Y 528.346,Z 284.769,A -85,B 0,C 180,E1 -11473.23,E2 -11473.23} C_VEL
LIN {X 0,Y 520.091,Z 265.604,A -85,B 0,C 180,E1 -11475.589,E2 -11475.589} C_VEL
LIN {X 0,Y 511.867,Z 248.983,A -85,B 0,C 180,E1 -11477.78,E2 -11477.78} C_VEL
LIN {X 0,Y 505.146,Z 236.611,A -85,B 0,C 180,E1 -11479.515,E2 -11479.515} C_VEL
LIN {X 0,Y 502.582,Z 232.134,A -85,B 0,C 180,E1 -11480.162,E2 -11480.162} C_VEL
LIN {X 0,Y 500.537,Z 228.181,A -85,B 0,C 180,E1 -11480.709,E2 -11480.709} C_VEL
LIN {X 0,Y 498.69,Z 225.789,A -85,B 0,C 180,E1 -11481.128,E2 -11481.128} C_VEL
LIN {X 0,Y 497.917,Z 223.213,A -85,B 0,C 180,E1 -11481.441,E2 -11481.441} C_VEL
LIN {X 0,Y 497.916,Z 223.21,A -85,B 0,C 180,E1 -11485.087,E2 -11485.087} C_VEL
LIN {X 0,Y 497.931,Z 223.201,A -85,B 0,C 180,E1 -11488.661,E2 -11488.661} C_VEL
LIN {X 0,Y 497.921,Z 223.181,A -85,B 0,C 180,E1 -11492.232,E2 -11492.232} C_VEL
LIN {X 0,Y 497.924,Z 223.174,A -85,B 0,C 180,E1 -11495.817,E2 -11495.817} C_VEL
LIN {X 0,Y 497.923,Z 223.206,A -85,B 0,C 180,E1 -11499.355,E2 -11499.355} C_VEL
LIN {X 0,Y 497.924,Z 223.176,A -85,B 0,C 180,E1 -11502.951,E2 -11502.951} C_VEL
LIN {X 0,Y 497.914,Z 223.184,A -85,B 0,C 180,E1 -11506.411,E2 -11506.411} C_VEL
LIN {X 0,Y 497.919,Z 223.2,A -85,B 0,C 180,E1 -11510.055,E2 -11510.055} C_VEL
LIN {X 0,Y 497.924,Z 223.166,A -85,B 0,C 180,E1 -11513.543,E2 -11513.543} C_VEL
LIN {X 0,Y 497.926,Z 223.205,A -85,B 0,C 180,E1 -11517.122,E2 -11517.122} C_VEL
LIN {X 0,Y 497.905,Z 223.163,A -85,B 0,C 180,E1 -11520.575,E2 -11520.575} C_VEL
LIN {X 0,Y 497.911,Z 223.208,A -85,B 0,C 180,E1 -11524.146,E2 -11524.146} C_VEL
LIN {X 0,Y 497.927,Z 223.163,A -85,B 0,C 180,E1 -11527.732,E2 -11527.732} C_VEL
LIN {X 0,Y 497.93,Z 223.205,A -85,B 0,C 180,E1 -11531.35,E2 -11531.35} C_VEL
LIN {X 0,Y 497.908,Z 223.202,A -85,B 0,C 180,E1 -11534.895,E2 -11534.895} C_VEL
LIN {X 0,Y 497.901,Z 223.2,A -85,B 0,C 180,E1 -11538.378,E2 -11538.378} C_VEL
LIN {X 0,Y 497.926,Z 223.2,A -85,B 0,C 180,E1 -11541.932,E2 -11541.932} C_VEL
LIN {X 0,Y 497.932,Z 223.207,A -85,B 0,C 180,E1 -11545.451,E2 -11545.451} C_VEL
LIN {X 0,Y 497.904,Z 223.202,A -85,B 0,C 180,E1 -11548.946,E2 -11548.946} C_VEL
LIN {X 0,Y 497.895,Z 223.235,A -85,B 0,C 180,E1 -11550.536,E2 -11550.536} C_VEL
LIN {X 0,Y 498.983,Z 226.339,A -85,B 0,C 180,E1 -11550.997,E2 -11550.997} C_VEL
LIN {X 0,Y 500.209,Z 227.869,A -85,B 0,C 180,E1 -11551.314,E2 -11551.314} C_VEL
LIN {X 0,Y 502.184,Z 232.043,A -85,B 0,C 180,E1 -11551.983,E2 -11551.983} C_VEL
LIN {X 0,Y 511.698,Z 250.645,A -85,B 0,C 180,E1 -11554.928,E2 -11554.928} C_VEL
LIN {X 0,Y 521.909,Z 270.924,A -85,B 0,C 180,E1 -11557.878,E2 -11557.878} C_VEL
LIN {X 0,Y 533.419,Z 294.639,A -85,B 0,C 180,E1 -11561.001,E2 -11561.001} C_VEL
LIN {X 0,Y 541.259,Z 311.648,A -85,B 0,C 180,E1 -11563.037,E2 -11563.037} C_VEL
LIN {X 0,Y 540.884,Z 316.257,A -85,B 0,C 180,E1 -11563.292,E2 -11563.292} C_VEL
LIN {X 0,Y 543.669,Z 344.055,A -85,B 0,C 180,E1 -11564.075,E2 -11564.075} C_VEL
LIN {X 0,Y 534.333,Z 582.812,A -85,B 0,C 180,E1 -11567.883,E2 -11567.883} C_VEL
LIN {X 0,Y 530.588,Z 692.929,A -85,B 0,C 180,E1 -11569.609,E2 -11569.609} C_VEL
LIN {X 0,Y 528.963,Z 717.488,A -85,B 0,C 180,E1 -11570.174,E2 -11570.174} C_VEL
LIN {X 0,Y 527.05,Z 741.067,A -85,B 0,C 180,E1 -11570.89,E2 -11570.89} C_VEL
LIN {X 0,Y 524.741,Z 763.853,A -85,B 0,C 180,E1 -11571.783,E2 -11571.783} C_VEL
LIN {X 0,Y 522.207,Z 786.241,A -85,B 0,C 180,E1 -11572.836,E2 -11572.836} C_VEL
LIN {X 0,Y 519.472,Z 807.492,A -85,B 0,C 180,E1 -11574.051,E2 -11574.051} C_VEL
LIN {X 0,Y 516.575,Z 828.598,A -85,B 0,C 180,E1 -11575.449,E2 -11575.449} C_VEL
LIN {X 0,Y 513.566,Z 849.024,A -85,B 0,C 180,E1 -11577.05,E2 -11577.05} C_VEL
LIN {X 0,Y 510.552,Z 869.166,A -85,B 0,C 180,E1 -11578.867,E2 -11578.867} C_VEL
LIN {X 0,Y 507.908,Z 886.18,A -85,B 0,C 180,E1 -11580.647,E2 -11580.647} C_VEL
LIN {X 0,Y 505.186,Z 904.141,A -85,B 0,C 180,E1 -11582.793,E2 -11582.793} C_VEL
LIN {X 0,Y 503.016,Z 918.875,A -85,B 0,C 180,E1 -11584.825,E2 -11584.825} C_VEL
LIN {X 0,Y 501.019,Z 933.36,A -85,B 0,C 180,E1 -11587.098,E2 -11587.098} C_VEL
LIN {X 0,Y 499.372,Z 946.381,A -85,B 0,C 180,E1 -11589.488,E2 -11589.488} C_VEL
LIN {X 0,Y 498.108,Z 958.222,A -85,B 0,C 180,E1 -11591.993,E2 -11591.993} C_VEL
LIN {X 0,Y 497.216,Z 968.061,A -85,B 0,C 180,E1 -11594.487,E2 -11594.487} C_VEL
LIN {X 0,Y 496.64,Z 976.729,A -85,B 0,C 180,E1 -11597.087,E2 -11597.087} C_VEL
LIN {X 0,Y 496.324,Z 983.79,A -85,B 0,C 180,E1 -11599.788,E2 -11599.788} C_VEL
LIN {X 0,Y 496.196,Z 988.809,A -85,B 0,C 180,E1 -11602.241,E2 -11602.241} C_VEL
LIN {X 0,Y 496.201,Z 992.633,A -85,B 0,C 180,E1 -11604.913,E2 -11604.913} C_VEL
LIN {X 0,Y 496.232,Z 994.538,A -85,B 0,C 180,E1 -11607.113,E2 -11607.113} C_VEL
LIN {X 0,Y 496.261,Z 995.356,A -85,B 0,C 180,E1 -11609.307,E2 -11609.307} C_VEL
LIN {X 0,Y 496.28,Z 994.989,A -85,B 0,C 180,E1 -11611.847,E2 -11611.847} C_VEL
LIN {X 0,Y 496.266,Z 992.974,A -85,B 0,C 180,E1 -11614.391,E2 -11614.391} C_VEL
LIN {X 0,Y 496.267,Z 989.888,A -85,B 0,C 180,E1 -11616.711,E2 -11616.711} C_VEL
LIN {X 0,Y 496.332,Z 984.812,A -85,B 0,C 180,E1 -11619.392,E2 -11619.392} C_VEL
LIN {X 0,Y 496.549,Z 978.157,A -85,B 0,C 180,E1 -11621.971,E2 -11621.971} C_VEL
LIN {X 0,Y 496.949,Z 970.715,A -85,B 0,C 180,E1 -11624.329,E2 -11624.329} C_VEL
LIN {X 0,Y 497.723,Z 960.221,A -85,B 0,C 180,E1 -11627.056,E2 -11627.056} C_VEL
LIN {X 0,Y 498.668,Z 949.927,A -85,B 0,C 180,E1 -11629.32,E2 -11629.32} C_VEL
LIN {X 0,Y 500.185,Z 935.955,A -85,B 0,C 180,E1 -11631.952,E2 -11631.952} C_VEL
LIN {X 0,Y 501.854,Z 922.46,A -85,B 0,C 180,E1 -11634.144,E2 -11634.144} C_VEL
LIN {X 0,Y 504.143,Z 905.307,A -85,B 0,C 180,E1 -11636.556,E2 -11636.556} C_VEL
LIN {X 0,Y 506.492,Z 888.608,A -85,B 0,C 180,E1 -11638.603,E2 -11638.603} C_VEL
LIN {X 0,Y 509.252,Z 869.46,A -85,B 0,C 180,E1 -11640.632,E2 -11640.632} C_VEL
LIN {X 0,Y 512.045,Z 850.249,A -85,B 0,C 180,E1 -11642.414,E2 -11642.414} C_VEL
LIN {X 0,Y 514.947,Z 829.398,A -85,B 0,C 180,E1 -11644.069,E2 -11644.069} C_VEL
LIN {X 0,Y 517.868,Z 808.115,A -85,B 0,C 180,E1 -11645.533,E2 -11645.533} C_VEL
LIN {X 0,Y 520.458,Z 787.463,A -85,B 0,C 180,E1 -11646.736,E2 -11646.736} C_VEL
LIN {X 0,Y 523.114,Z 765.032,A -85,B 0,C 180,E1 -11647.848,E2 -11647.848} C_VEL
LIN {X 0,Y 525.438,Z 742.393,A -85,B 0,C 180,E1 -11648.761,E2 -11648.761} C_VEL
LIN {X 0,Y 527.646,Z 716.844,A -85,B 0,C 180,E1 -11649.58,E2 -11649.58} C_VEL
LIN {X 0,Y 529.391,Z 692.114,A -85,B 0,C 180,E1 -11650.167,E2 -11650.167} C_VEL
LIN {X 0,Y 534.165,Z 581.206,A -85,B 0,C 180,E1 -11652.032,E2 -11652.032} C_VEL
LIN {X 0,Y 538.929,Z 503.389,A -85,B 0,C 180,E1 -11653.48,E2 -11653.48} C_VEL
LIN {X 0,Y 545.076,Z 430.601,A -85,B 0,C 180,E1 -11654.954,E2 -11654.954} C_VEL
LIN {X 0,Y 552.742,Z 362.529,A -85,B 0,C 180,E1 -11656.419,E2 -11656.419} C_VEL
LIN {X 0,Y 554.177,Z 352.559,A -85,B 0,C 180,E1 -11656.646,E2 -11656.646} C_VEL
LIN {X 0,Y 556.507,Z 348.629,A -85,B 0,C 180,E1 -11656.842,E2 -11656.842} C_VEL
LIN {X 0,Y 564.301,Z 335.308,A -85,B 0,C 180,E1 -11658.132,E2 -11658.132} C_VEL
LIN {X 0,Y 554.245,Z 350.827,A -85,B 0,C 180,E1 -11659.905,E2 -11659.905} C_VEL
LIN {X 0,Y 545.277,Z 369.18,A -85,B 0,C 180,E1 -11661.876,E2 -11661.876} C_VEL
LIN {X 0,Y 541.272,Z 380.071,A -85,B 0,C 180,E1 -11662.971,E2 -11662.971} C_VEL
LIN {X 0,Y 539.882,Z 395.489,A -85,B 0,C 180,E1 -11664.189,E2 -11664.189} C_VEL
LIN {X 0,Y 538.901,Z 414.359,A -85,B 0,C 180,E1 -11665.508,E2 -11665.508} C_VEL
LIN {X 0,Y 538.23,Z 436.085,A -85,B 0,C 180,E1 -11666.823,E2 -11666.823} C_VEL
LIN {X 0,Y 537.746,Z 462.687,A -85,B 0,C 180,E1 -11668.233,E2 -11668.233} C_VEL
LIN {X 0,Y 537.226,Z 494.399,A -85,B 0,C 180,E1 -11669.678,E2 -11669.678} C_VEL
LIN {X 0,Y 536.808,Z 507.507,A -85,B 0,C 180,E1 -11670.196,E2 -11670.196} C_VEL
LIN {X 0,Y 525.195,Z 612.307,A -85,B 0,C 180,E1 -11672.865,E2 -11672.865} C_VEL
LIN {X 0,Y 518.134,Z 690.947,A -85,B 0,C 180,E1 -11674.889,E2 -11674.889} C_VEL
LIN {X 0,Y 515.856,Z 715.335,A -85,B 0,C 180,E1 -11675.737,E2 -11675.737} C_VEL
LIN {X 0,Y 513.695,Z 737.418,A -85,B 0,C 180,E1 -11676.726,E2 -11676.726} C_VEL
LIN {X 0,Y 511.583,Z 758.559,A -85,B 0,C 180,E1 -11677.886,E2 -11677.886} C_VEL
LIN {X 0,Y 509.453,Z 778.751,A -85,B 0,C 180,E1 -11679.252,E2 -11679.252} C_VEL
LIN {X 0,Y 507.637,Z 795.554,A -85,B 0,C 180,E1 -11680.616,E2 -11680.616} C_VEL
LIN {X 0,Y 505.847,Z 811.517,A -85,B 0,C 180,E1 -11682.159,E2 -11682.159} C_VEL
LIN {X 0,Y 504.229,Z 825.364,A -85,B 0,C 180,E1 -11683.763,E2 -11683.763} C_VEL
LIN {X 0,Y 502.759,Z 837.804,A -85,B 0,C 180,E1 -11685.488,E2 -11685.488} C_VEL
LIN {X 0,Y 501.427,Z 848.665,A -85,B 0,C 180,E1 -11687.329,E2 -11687.329} C_VEL
LIN {X 0,Y 500.343,Z 857.501,A -85,B 0,C 180,E1 -11689.173,E2 -11689.173} C_VEL
LIN {X 0,Y 499.418,Z 864.812,A -85,B 0,C 180,E1 -11691.132,E2 -11691.132} C_VEL
LIN {X 0,Y 498.69,Z 870.567,A -85,B 0,C 180,E1 -11693.206,E2 -11693.206} C_VEL
LIN {X 0,Y 498.146,Z 874.376,A -85,B 0,C 180,E1 -11695.279,E2 -11695.279} C_VEL
LIN {X 0,Y 497.766,Z 876.362,A -85,B 0,C 180,E1 -11697.352,E2 -11697.352} C_VEL
LIN {X 0,Y 497.53,Z 876.601,A -85,B 0,C 180,E1 -11699.424,E2 -11699.424} C_VEL
LIN {X 0,Y 497.397,Z 875.104,A -85,B 0,C 180,E1 -11701.498,E2 -11701.498} C_VEL
LIN {X 0,Y 497.377,Z 871.889,A -85,B 0,C 180,E1 -11703.573,E2 -11703.573} C_VEL
LIN {X 0,Y 497.487,Z 866.903,A -85,B 0,C 180,E1 -11705.652,E2 -11705.652} C_VEL
LIN {X 0,Y 497.726,Z 860.486,A -85,B 0,C 180,E1 -11707.619,E2 -11707.619} C_VEL
LIN {X 0,Y 498.141,Z 852.263,A -85,B 0,C 180,E1 -11709.59,E2 -11709.59} C_VEL
LIN {X 0,Y 498.775,Z 842.028,A -85,B 0,C 180,E1 -11711.564,E2 -11711.564} C_VEL
LIN {X 0,Y 499.598,Z 830.284,A -85,B 0,C 180,E1 -11713.424,E2 -11713.424} C_VEL
LIN {X 0,Y 500.6,Z 817.064,A -85,B 0,C 180,E1 -11715.169,E2 -11715.169} C_VEL
LIN {X 0,Y 501.788,Z 802.012,A -85,B 0,C 180,E1 -11716.832,E2 -11716.832} C_VEL
LIN {X 0,Y 503.112,Z 785.453,A -85,B 0,C 180,E1 -11718.361,E2 -11718.361} C_VEL
LIN {X 0,Y 504.503,Z 767.326,A -85,B 0,C 180,E1 -11719.75,E2 -11719.75} C_VEL
LIN {X 0,Y 505.928,Z 747.989,A -85,B 0,C 180,E1 -11720.96,E2 -11720.96} C_VEL
LIN {X 0,Y 507.242,Z 728.723,A -85,B 0,C 180,E1 -11721.935,E2 -11721.935} C_VEL
LIN {X 0,Y 508.498,Z 707.478,A -85,B 0,C 180,E1 -11722.774,E2 -11722.774} C_VEL
LIN {X 0,Y 509.582,Z 686,A -85,B 0,C 180,E1 -11723.397,E2 -11723.397} C_VEL
LIN {X 0,Y 510.841,Z 649.884,A -85,B 0,C 180,E1 -11724.097,E2 -11724.097} C_VEL
LIN {X 0,Y 516.396,Z 497.59,A -85,B 0,C 180,E1 -11726.908,E2 -11726.908} C_VEL
LIN {X 0,Y 511.577,Z 447.124,A -85,B 0,C 180,E1 -11728.261,E2 -11728.261} C_VEL
LIN {X 0,Y 515.756,Z 394.023,A -85,B 0,C 180,E1 -11732.091,E2 -11732.091} C_VEL
LIN {X 0,Y 519.879,Z 347.002,A -85,B 0,C 180,E1 -11735.51,E2 -11735.51} C_VEL
LIN {X 0,Y 524.881,Z 295.349,A -85,B 0,C 180,E1 -11739.302,E2 -11739.302} C_VEL
LIN {X 0,Y 525.082,Z 291.057,A -85,B 0,C 180,E1 -11739.638,E2 -11739.638} C_VEL
LIN {X 0,Y 516.748,Z 268.716,A -85,B 0,C 180,E1 -11742.178,E2 -11742.178} C_VEL
LIN {X 0,Y 513.337,Z 259.733,A -85,B 0,C 180,E1 -11743.286,E2 -11743.286} C_VEL
LIN {X 0,Y 515.183,Z 260.362,A -85,B 0,C 180,E1 -11743.551,E2 -11743.551} C_VEL
LIN {X 0,Y 517.808,Z 260.741,A -85,B 0,C 180,E1 -11743.887,E2 -11743.887} C_VEL
LIN {X 0,Y 525.294,Z 277.616,A -85,B 0,C 180,E1 -11746.015,E2 -11746.015} C_VEL
LIN {X 0,Y 532.91,Z 297.004,A -85,B 0,C 180,E1 -11748.311,E2 -11748.311} C_VEL
LIN {X 0,Y 536.205,Z 306.454,A -85,B 0,C 180,E1 -11749.373,E2 -11749.373} C_VEL
LIN {X 0,Y 535.707,Z 348.21,A -85,B 0,C 180,E1 -11752.251,E2 -11752.251} C_VEL
LIN {X 0,Y 535.539,Z 354.533,A -85,B 0,C 180,E1 -11752.641,E2 -11752.641} C_VEL
LIN {X 0,Y 532.735,Z 368.037,A -85,B 0,C 180,E1 -11753.145,E2 -11753.145} C_VEL
LIN {X 0,Y 531.147,Z 420.838,A -85,B 0,C 180,E1 -11753.918,E2 -11753.918} C_VEL
LIN {X 0,Y 530.074,Z 428.519,A -85,B 0,C 180,E1 -11753.968,E2 -11753.968} C_VEL
LIN {X 0,Y 524.319,Z 448.958,A -85,B 0,C 180,E1 -11753.874,E2 -11753.874} C_VEL
LIN {X 0,Y 523.463,Z 455.536,A -85,B 0,C 180,E1 -11753.934,E2 -11753.934} C_VEL
LIN {X 0,Y 519.987,Z 527.674,A -85,B 0,C 180,E1 -11755.214,E2 -11755.214} C_VEL
LIN {X 0,Y 515.254,Z 607.323,A -85,B 0,C 180,E1 -11756.843,E2 -11756.843} C_VEL
LIN {X 0,Y 513.124,Z 648.267,A -85,B 0,C 180,E1 -11757.815,E2 -11757.815} C_VEL
LIN {X 0,Y 511.85,Z 670.06,A -85,B 0,C 180,E1 -11758.529,E2 -11758.529} C_VEL
LIN {X 0,Y 510.196,Z 691.298,A -85,B 0,C 180,E1 -11759.431,E2 -11759.431} C_VEL
LIN {X 0,Y 508.197,Z 712.118,A -85,B 0,C 180,E1 -11760.536,E2 -11760.536} C_VEL
LIN {X 0,Y 506.025,Z 731.949,A -85,B 0,C 180,E1 -11761.819,E2 -11761.819} C_VEL
LIN {X 0,Y 503.772,Z 750.161,A -85,B 0,C 180,E1 -11763.221,E2 -11763.221} C_VEL
LIN {X 0,Y 501.33,Z 768.422,A -85,B 0,C 180,E1 -11764.89,E2 -11764.89} C_VEL
LIN {X 0,Y 498.97,Z 785.034,A -85,B 0,C 180,E1 -11766.686,E2 -11766.686} C_VEL
LIN {X 0,Y 496.886,Z 799.497,A -85,B 0,C 180,E1 -11768.516,E2 -11768.516} C_VEL
LIN {X 0,Y 494.823,Z 813.874,A -85,B 0,C 180,E1 -11770.646,E2 -11770.646} C_VEL
LIN {X 0,Y 493.063,Z 826.677,A -85,B 0,C 180,E1 -11772.899,E2 -11772.899} C_VEL
LIN {X 0,Y 491.688,Z 837.411,A -85,B 0,C 180,E1 -11775.153,E2 -11775.153} C_VEL
LIN {X 0,Y 490.619,Z 846.749,A -85,B 0,C 180,E1 -11777.524,E2 -11777.524} C_VEL
LIN {X 0,Y 489.836,Z 854.52,A -85,B 0,C 180,E1 -11780.008,E2 -11780.008} C_VEL
LIN {X 0,Y 489.348,Z 860.2,A -85,B 0,C 180,E1 -11782.368,E2 -11782.368} C_VEL
LIN {X 0,Y 489.076,Z 864.511,A -85,B 0,C 180,E1 -11784.839,E2 -11784.839} C_VEL
LIN {X 0,Y 488.935,Z 867.192,A -85,B 0,C 180,E1 -11787.304,E2 -11787.304} C_VEL
LIN {X 0,Y 488.889,Z 868.168,A -85,B 0,C 180,E1 -11789.766,E2 -11789.766} C_VEL
LIN {X 0,Y 488.916,Z 867.511,A -85,B 0,C 180,E1 -11792.227,E2 -11792.227} C_VEL
LIN {X 0,Y 489.04,Z 865.259,A -85,B 0,C 180,E1 -11794.691,E2 -11794.691} C_VEL
LIN {X 0,Y 489.284,Z 861.392,A -85,B 0,C 180,E1 -11797.161,E2 -11797.161} C_VEL
LIN {X 0,Y 489.72,Z 855.73,A -85,B 0,C 180,E1 -11799.638,E2 -11799.638} C_VEL
LIN {X 0,Y 490.421,Z 848.634,A -85,B 0,C 180,E1 -11802.003,E2 -11802.003} C_VEL
LIN {X 0,Y 491.458,Z 839.295,A -85,B 0,C 180,E1 -11804.492,E2 -11804.492} C_VEL
LIN {X 0,Y 492.775,Z 828.984,A -85,B 0,C 180,E1 -11806.746,E2 -11806.746} C_VEL
LIN {X 0,Y 494.367,Z 817.386,A -85,B 0,C 180,E1 -11808.881,E2 -11808.881} C_VEL
LIN {X 0,Y 496.446,Z 802.797,A -85,B 0,C 180,E1 -11811.132,E2 -11811.132} C_VEL
LIN {X 0,Y 498.742,Z 786.853,A -85,B 0,C 180,E1 -11813.2,E2 -11813.2} C_VEL
LIN {X 0,Y 501.156,Z 769.789,A -85,B 0,C 180,E1 -11815.067,E2 -11815.067} C_VEL
LIN {X 0,Y 503.469,Z 752.531,A -85,B 0,C 180,E1 -11816.669,E2 -11816.669} C_VEL
LIN {X 0,Y 505.808,Z 733.895,A -85,B 0,C 180,E1 -11818.136,E2 -11818.136} C_VEL
LIN {X 0,Y 508.074,Z 713.598,A -85,B 0,C 180,E1 -11819.472,E2 -11819.472} C_VEL
LIN {X 0,Y 510.065,Z 693.123,A -85,B 0,C 180,E1 -11820.577,E2 -11820.577} C_VEL
LIN {X 0,Y 511.731,Z 672.225,A -85,B 0,C 180,E1 -11821.487,E2 -11821.487} C_VEL
LIN {X 0,Y 513.065,Z 650.65,A -85,B 0,C 180,E1 -11822.216,E2 -11822.216} C_VEL
LIN {X 0,Y 515.022,Z 611.532,A -85,B 0,C 180,E1 -11823.162,E2 -11823.162} C_VEL
LIN {X 0,Y 519.861,Z 530.594,A -85,B 0,C 180,E1 -11824.825,E2 -11824.825} C_VEL
LIN {X 0,Y 523.366,Z 458.843,A -85,B 0,C 180,E1 -11826.107,E2 -11826.107} C_VEL
LIN {X 0,Y 526.252,Z 374.974,A -85,B 0,C 180,E1 -11827.384,E2 -11827.384} C_VEL
LIN {X 0,Y 526.568,Z 369.122,A -85,B 0,C 180,E1 -11827.488,E2 -11827.488} C_VEL
LIN {X 0,Y 529.673,Z 354.611,A -85,B 0,C 180,E1 -11828.076,E2 -11828.076} C_VEL
LIN {X 0,Y 529.967,Z 316.559,A -85,B 0,C 180,E1 -11830.671,E2 -11830.671} C_VEL
LIN {X 0,Y 529.934,Z 309.573,A -85,B 0,C 180,E1 -11831.186,E2 -11831.186} C_VEL
LIN {X 0,Y 522.461,Z 289.382,A -85,B 0,C 180,E1 -11833.549,E2 -11833.549} C_VEL
LIN {X 0,Y 513.927,Z 269.463,A -85,B 0,C 180,E1 -11836.044,E2 -11836.044} C_VEL
LIN {X 0,Y 505.067,Z 251.535,A -85,B 0,C 180,E1 -11838.455,E2 -11838.455} C_VEL
LIN {X 0,Y 497.989,Z 238.548,A -85,B 0,C 180,E1 -11840.32,E2 -11840.32} C_VEL
LIN {X 0,Y 495.018,Z 233.573,A -85,B 0,C 180,E1 -11841.083,E2 -11841.083} C_VEL
LIN {X 0,Y 492.968,Z 229.775,A -85,B 0,C 180,E1 -11841.635,E2 -11841.635} C_VEL
LIN {X 0,Y 490.723,Z 226.675,A -85,B 0,C 180,E1 -11842.17,E2 -11842.17} C_VEL
LIN {X 0,Y 489.99,Z 224.177,A -85,B 0,C 180,E1 -11842.481,E2 -11842.481} C_VEL
LIN {X 0,Y 489.986,Z 224.18,A -85,B 0,C 180,E1 -11846.004,E2 -11846.004} C_VEL
LIN {X 0,Y 489.995,Z 224.192,A -85,B 0,C 180,E1 -11849.675,E2 -11849.675} C_VEL
LIN {X 0,Y 489.98,Z 224.188,A -85,B 0,C 180,E1 -11853.193,E2 -11853.193} C_VEL
LIN {X 0,Y 489.987,Z 224.157,A -85,B 0,C 180,E1 -11856.806,E2 -11856.806} C_VEL
LIN {X 0,Y 489.981,Z 224.179,A -85,B 0,C 180,E1 -11860.323,E2 -11860.323} C_VEL
LIN {X 0,Y 489.985,Z 224.184,A -85,B 0,C 180,E1 -11863.977,E2 -11863.977} C_VEL
LIN {X 0,Y 489.981,Z 224.153,A -85,B 0,C 180,E1 -11867.507,E2 -11867.507} C_VEL
LIN {X 0,Y 489.989,Z 224.194,A -85,B 0,C 180,E1 -11871.078,E2 -11871.078} C_VEL
LIN {X 0,Y 489.972,Z 224.156,A -85,B 0,C 180,E1 -11874.614,E2 -11874.614} C_VEL
LIN {X 0,Y 489.972,Z 224.189,A -85,B 0,C 180,E1 -11878.246,E2 -11878.246} C_VEL
LIN {X 0,Y 489.984,Z 224.161,A -85,B 0,C 180,E1 -11881.754,E2 -11881.754} C_VEL
LIN {X 0,Y 489.988,Z 224.178,A -85,B 0,C 180,E1 -11885.269,E2 -11885.269} C_VEL
LIN {X 0,Y 489.967,Z 224.171,A -85,B 0,C 180,E1 -11888.686,E2 -11888.686} C_VEL
LIN {X 0,Y 489.968,Z 224.198,A -85,B 0,C 180,E1 -11892.253,E2 -11892.253} C_VEL
LIN {X 0,Y 489.992,Z 224.186,A -85,B 0,C 180,E1 -11895.748,E2 -11895.748} C_VEL
LIN {X 0,Y 489.992,Z 224.189,A -85,B 0,C 180,E1 -11899.304,E2 -11899.304} C_VEL
LIN {X 0,Y 489.963,Z 224.2,A -85,B 0,C 180,E1 -11902.814,E2 -11902.814} C_VEL
LIN {X 0,Y 489.96,Z 224.191,A -85,B 0,C 180,E1 -11906.416,E2 -11906.416} C_VEL
LIN {X 0,Y 490.002,Z 224.209,A -85,B 0,C 180,E1 -11909.538,E2 -11909.538} C_VEL
LIN {X 0,Y 491.217,Z 227.578,A -85,B 0,C 180,E1 -11910.049,E2 -11910.049} C_VEL
LIN {X 0,Y 492.371,Z 229.242,A -85,B 0,C 180,E1 -11910.375,E2 -11910.375} C_VEL
LIN {X 0,Y 494.359,Z 233.153,A -85,B 0,C 180,E1 -11911.049,E2 -11911.049} C_VEL
LIN {X 0,Y 504.126,Z 252.236,A -85,B 0,C 180,E1 -11914.146,E2 -11914.146} C_VEL
LIN {X 0,Y 514.417,Z 272.721,A -85,B 0,C 180,E1 -11917.193,E2 -11917.193} C_VEL
LIN {X 0,Y 525.439,Z 295.438,A -85,B 0,C 180,E1 -11920.263,E2 -11920.263} C_VEL
LIN {X 0,Y 534.591,Z 314.923,A -85,B 0,C 180,E1 -11922.667,E2 -11922.667} C_VEL
LIN {X 0,Y 534.669,Z 318.06,A -85,B 0,C 180,E1 -11922.791,E2 -11922.791} C_VEL
LIN {X 0,Y 537.329,Z 345.264,A -85,B 0,C 180,E1 -11923.568,E2 -11923.568} C_VEL
LIN {X 0,Y 527.676,Z 580.872,A -85,B 0,C 180,E1 -11927.383,E2 -11927.383} C_VEL
LIN {X 0,Y 523.674,Z 692.969,A -85,B 0,C 180,E1 -11929.17,E2 -11929.17} C_VEL
LIN {X 0,Y 521.999,Z 717.336,A -85,B 0,C 180,E1 -11929.74,E2 -11929.74} C_VEL
LIN {X 0,Y 520.001,Z 741.084,A -85,B 0,C 180,E1 -11930.471,E2 -11930.471} C_VEL
LIN {X 0,Y 517.579,Z 764.203,A -85,B 0,C 180,E1 -11931.392,E2 -11931.392} C_VEL
LIN {X 0,Y 514.823,Z 787.471,A -85,B 0,C 180,E1 -11932.515,E2 -11932.515} C_VEL
LIN {X 0,Y 512.067,Z 808.281,A -85,B 0,C 180,E1 -11933.726,E2 -11933.726} C_VEL
LIN {X 0,Y 508.957,Z 830.059,A -85,B 0,C 180,E1 -11935.205,E2 -11935.205} C_VEL
LIN {X 0,Y 506.133,Z 848.679,A -85,B 0,C 180,E1 -11936.688,E2 -11936.688} C_VEL
LIN {X 0,Y 503.052,Z 868.567,A -85,B 0,C 180,E1 -11938.507,E2 -11938.507} C_VEL
LIN {X 0,Y 500.267,Z 885.971,A -85,B 0,C 180,E1 -11940.351,E2 -11940.351} C_VEL
LIN {X 0,Y 497.521,Z 903.473,A -85,B 0,C 180,E1 -11942.468,E2 -11942.468} C_VEL
LIN {X 0,Y 495.271,Z 918.206,A -85,B 0,C 180,E1 -11944.531,E2 -11944.531} C_VEL
LIN {X 0,Y 493.099,Z 933.397,A -85,B 0,C 180,E1 -11946.961,E2 -11946.961} C_VEL
LIN {X 0,Y 491.491,Z 945.773,A -85,B 0,C 180,E1 -11949.269,E2 -11949.269} C_VEL
LIN {X 0,Y 490.173,Z 957.591,A -85,B 0,C 180,E1 -11951.814,E2 -11951.814} C_VEL
LIN {X 0,Y 489.254,Z 967.431,A -85,B 0,C 180,E1 -11954.35,E2 -11954.35} C_VEL
LIN {X 0,Y 488.666,Z 976.092,A -85,B 0,C 180,E1 -11956.993,E2 -11956.993} C_VEL
LIN {X 0,Y 488.356,Z 982.848,A -85,B 0,C 180,E1 -11959.62,E2 -11959.62} C_VEL
LIN {X 0,Y 488.246,Z 987.67,A -85,B 0,C 180,E1 -11961.995,E2 -11961.995} C_VEL
LIN {X 0,Y 488.235,Z 991.624,A -85,B 0,C 180,E1 -11964.712,E2 -11964.712} C_VEL
LIN {X 0,Y 488.278,Z 993.657,A -85,B 0,C 180,E1 -11967.066,E2 -11967.066} C_VEL
LIN {X 0,Y 488.31,Z 994.473,A -85,B 0,C 180,E1 -11969.296,E2 -11969.296} C_VEL
LIN {X 0,Y 488.328,Z 994.095,A -85,B 0,C 180,E1 -11971.877,E2 -11971.877} C_VEL
LIN {X 0,Y 488.308,Z 992.061,A -85,B 0,C 180,E1 -11974.463,E2 -11974.463} C_VEL
LIN {X 0,Y 488.303,Z 988.949,A -85,B 0,C 180,E1 -11976.821,E2 -11976.821} C_VEL
LIN {X 0,Y 488.368,Z 983.837,A -85,B 0,C 180,E1 -11979.546,E2 -11979.546} C_VEL
LIN {X 0,Y 488.591,Z 977.137,A -85,B 0,C 180,E1 -11982.169,E2 -11982.169} C_VEL
LIN {X 0,Y 489.01,Z 969.667,A -85,B 0,C 180,E1 -11984.566,E2 -11984.566} C_VEL
LIN {X 0,Y 489.822,Z 959.11,A -85,B 0,C 180,E1 -11987.34,E2 -11987.34} C_VEL
LIN {X 0,Y 490.822,Z 948.79,A -85,B 0,C 180,E1 -11989.642,E2 -11989.642} C_VEL
LIN {X 0,Y 492.431,Z 934.759,A -85,B 0,C 180,E1 -11992.316,E2 -11992.316} C_VEL
LIN {X 0,Y 494.254,Z 920.678,A -85,B 0,C 180,E1 -11994.629,E2 -11994.629} C_VEL
LIN {X 0,Y 496.543,Z 904.403,A -85,B 0,C 180,E1 -11996.942,E2 -11996.942} C_VEL
LIN {X 0,Y 499.003,Z 887.809,A -85,B 0,C 180,E1 -11999.007,E2 -11999.007} C_VEL
LIN {X 0,Y 501.911,Z 868.716,A -85,B 0,C 180,E1 -12001.063,E2 -12001.063} C_VEL
LIN {X 0,Y 504.876,Z 849.322,A -85,B 0,C 180,E1 -12002.889,E2 -12002.889} C_VEL
LIN {X 0,Y 507.891,Z 828.825,A -85,B 0,C 180,E1 -12004.541,E2 -12004.541} C_VEL
LIN {X 0,Y 510.965,Z 807.693,A -85,B 0,C 180,E1 -12006.018,E2 -12006.018} C_VEL
LIN {X 0,Y 513.725,Z 786.842,A -85,B 0,C 180,E1 -12007.252,E2 -12007.252} C_VEL
LIN {X 0,Y 516.513,Z 764.639,A -85,B 0,C 180,E1 -12008.37,E2 -12008.37} C_VEL
LIN {X 0,Y 518.91,Z 742.736,A -85,B 0,C 180,E1 -12009.271,E2 -12009.271} C_VEL
LIN {X 0,Y 521.22,Z 718.185,A -85,B 0,C 180,E1 -12010.084,E2 -12010.084} C_VEL
LIN {X 0,Y 523.123,Z 693.188,A -85,B 0,C 180,E1 -12010.699,E2 -12010.699} C_VEL
LIN {X 0,Y 528.462,Z 583.74,A -85,B 0,C 180,E1 -12012.611,E2 -12012.611} C_VEL
LIN {X 0,Y 533.562,Z 509.512,A -85,B 0,C 180,E1 -12014.038,E2 -12014.038} C_VEL
LIN {X 0,Y 540.211,Z 438.406,A -85,B 0,C 180,E1 -12015.523,E2 -12015.523} C_VEL
LIN {X 0,Y 548.593,Z 370.874,A -85,B 0,C 180,E1 -12017.013,E2 -12017.013} C_VEL
LIN {X 0,Y 550.864,Z 355.837,A -85,B 0,C 180,E1 -12017.357,E2 -12017.357} C_VEL
LIN {X 0,Y 553.527,Z 351.611,A -85,B 0,C 180,E1 -12017.554,E2 -12017.554} C_VEL
LIN {X 0,Y 557.392,Z 345.328,A -85,B 0,C 180,E1 -12018.174,E2 -12018.174} C_VEL
LIN {X 0,Y 547.265,Z 361.034,A -85,B 0,C 180,E1 -12019.974,E2 -12019.974} C_VEL
LIN {X 0,Y 541.273,Z 373.163,A -85,B 0,C 180,E1 -12021.278,E2 -12021.278} C_VEL
LIN {X 0,Y 538.529,Z 389.206,A -85,B 0,C 180,E1 -12022.684,E2 -12022.684} C_VEL
LIN {X 0,Y 536.557,Z 407.669,A -85,B 0,C 180,E1 -12024.109,E2 -12024.109} C_VEL
LIN {X 0,Y 535.061,Z 430.229,A -85,B 0,C 180,E1 -12025.61,E2 -12025.61} C_VEL
LIN {X 0,Y 533.805,Z 458.593,A -85,B 0,C 180,E1 -12027.217,E2 -12027.217} C_VEL
LIN {X 0,Y 532.714,Z 490.752,A -85,B 0,C 180,E1 -12028.767,E2 -12028.767} C_VEL
LIN {X 0,Y 531.971,Z 508.887,A -85,B 0,C 180,E1 -12029.526,E2 -12029.526} C_VEL
LIN {X 0,Y 519.156,Z 616.895,A -85,B 0,C 180,E1 -12032.348,E2 -12032.348} C_VEL
LIN {X 0,Y 512.023,Z 690.774,A -85,B 0,C 180,E1 -12034.304,E2 -12034.304} C_VEL
LIN {X 0,Y 509.623,Z 714.531,A -85,B 0,C 180,E1 -12035.142,E2 -12035.142} C_VEL
LIN {X 0,Y 507.126,Z 738.308,A -85,B 0,C 180,E1 -12036.221,E2 -12036.221} C_VEL
LIN {X 0,Y 504.819,Z 759.265,A -85,B 0,C 180,E1 -12037.402,E2 -12037.402} C_VEL
LIN {X 0,Y 502.66,Z 778.514,A -85,B 0,C 180,E1 -12038.714,E2 -12038.714} C_VEL
LIN {X 0,Y 500.462,Z 797.298,A -85,B 0,C 180,E1 -12040.266,E2 -12040.266} C_VEL
LIN {X 0,Y 498.615,Z 812.524,A -85,B 0,C 180,E1 -12041.77,E2 -12041.77} C_VEL
LIN {X 0,Y 496.895,Z 826.413,A -85,B 0,C 180,E1 -12043.397,E2 -12043.397} C_VEL
LIN {X 0,Y 495.3,Z 838.799,A -85,B 0,C 180,E1 -12045.144,E2 -12045.144} C_VEL
LIN {X 0,Y 493.962,Z 849.119,A -85,B 0,C 180,E1 -12046.896,E2 -12046.896} C_VEL
LIN {X 0,Y 492.693,Z 858.533,A -85,B 0,C 180,E1 -12048.884,E2 -12048.884} C_VEL
LIN {X 0,Y 491.695,Z 865.896,A -85,B 0,C 180,E1 -12050.873,E2 -12050.873} C_VEL
LIN {X 0,Y 490.924,Z 871.352,A -85,B 0,C 180,E1 -12052.863,E2 -12052.863} C_VEL
LIN {X 0,Y 490.35,Z 875.114,A -85,B 0,C 180,E1 -12054.852,E2 -12054.852} C_VEL
LIN {X 0,Y 489.918,Z 877.331,A -85,B 0,C 180,E1 -12056.958,E2 -12056.958} C_VEL
LIN {X 0,Y 489.633,Z 877.765,A -85,B 0,C 180,E1 -12059.064,E2 -12059.064} C_VEL
LIN {X 0,Y 489.477,Z 876.465,A -85,B 0,C 180,E1 -12061.171,E2 -12061.171} C_VEL
LIN {X 0,Y 489.433,Z 873.448,A -85,B 0,C 180,E1 -12063.279,E2 -12063.279} C_VEL
LIN {X 0,Y 489.52,Z 868.653,A -85,B 0,C 180,E1 -12065.391,E2 -12065.391} C_VEL
LIN {X 0,Y 489.765,Z 862.002,A -85,B 0,C 180,E1 -12067.508,E2 -12067.508} C_VEL
LIN {X 0,Y 490.208,Z 853.338,A -85,B 0,C 180,E1 -12069.628,E2 -12069.628} C_VEL
LIN {X 0,Y 490.861,Z 843.095,A -85,B 0,C 180,E1 -12071.634,E2 -12071.634} C_VEL
LIN {X 0,Y 491.709,Z 831.353,A -85,B 0,C 180,E1 -12073.524,E2 -12073.524} C_VEL
LIN {X 0,Y 492.741,Z 818.133,A -85,B 0,C 180,E1 -12075.296,E2 -12075.296} C_VEL
LIN {X 0,Y 493.933,Z 803.449,A -85,B 0,C 180,E1 -12076.948,E2 -12076.948} C_VEL
LIN {X 0,Y 495.268,Z 787.239,A -85,B 0,C 180,E1 -12078.48,E2 -12078.48} C_VEL
LIN {X 0,Y 496.696,Z 769.35,A -85,B 0,C 180,E1 -12079.89,E2 -12079.89} C_VEL
LIN {X 0,Y 498.155,Z 750.407,A -85,B 0,C 180,E1 -12081.118,E2 -12081.118} C_VEL
LIN {X 0,Y 499.578,Z 730.331,A -85,B 0,C 180,E1 -12082.165,E2 -12082.165} C_VEL
LIN {X 0,Y 500.861,Z 709.536,A -85,B 0,C 180,E1 -12083.015,E2 -12083.015} C_VEL
LIN {X 0,Y 501.993,Z 688.039,A -85,B 0,C 180,E1 -12083.667,E2 -12083.667} C_VEL
LIN {X 0,Y 503.092,Z 659.124,A -85,B 0,C 180,E1 -12084.258,E2 -12084.258} C_VEL
LIN {X 0,Y 509.188,Z 498.647,A -85,B 0,C 180,E1 -12087.28,E2 -12087.28} C_VEL
LIN {X 0,Y 504.307,Z 446.424,A -85,B 0,C 180,E1 -12088.706,E2 -12088.706} C_VEL
LIN {X 0,Y 508.678,Z 393.244,A -85,B 0,C 180,E1 -12092.588,E2 -12092.588} C_VEL
LIN {X 0,Y 513.168,Z 344.374,A -85,B 0,C 180,E1 -12096.185,E2 -12096.185} C_VEL
LIN {X 0,Y 518.183,Z 294.693,A -85,B 0,C 180,E1 -12099.875,E2 -12099.875} C_VEL
LIN {X 0,Y 510.877,Z 274.648,A -85,B 0,C 180,E1 -12102.169,E2 -12102.169} C_VEL
LIN {X 0,Y 507.832,Z 266.752,A -85,B 0,C 180,E1 -12103.135,E2 -12103.135} C_VEL
LIN {X 0,Y 510.169,Z 267.426,A -85,B 0,C 180,E1 -12103.467,E2 -12103.467} C_VEL
LIN {X 0,Y 513.169,Z 267.803,A -85,B 0,C 180,E1 -12103.851,E2 -12103.851} C_VEL
LIN {X 0,Y 521.029,Z 285.994,A -85,B 0,C 180,E1 -12106.149,E2 -12106.149} C_VEL
LIN {X 0,Y 528.966,Z 307.024,A -85,B 0,C 180,E1 -12108.629,E2 -12108.629} C_VEL
LIN {X 0,Y 530.034,Z 310.339,A -85,B 0,C 180,E1 -12108.99,E2 -12108.99} C_VEL
LIN {X 0,Y 529.565,Z 353.244,A -85,B 0,C 180,E1 -12111.939,E2 -12111.939} C_VEL
LIN {X 0,Y 529.287,Z 356.557,A -85,B 0,C 180,E1 -12112.123,E2 -12112.123} C_VEL
LIN {X 0,Y 526.333,Z 370.703,A -85,B 0,C 180,E1 -12112.651,E2 -12112.651} C_VEL
LIN {X 0,Y 523.463,Z 455.536,A -85,B 0,C 180,E1 -12113.934,E2 -12113.934} C_VEL
LIN {X 0,Y 522.35,Z 463.2,A -85,B 0,C 180,E1 -12113.996,E2 -12113.996} C_VEL
LIN {X 0,Y 516.416,Z 483.598,A -85,B 0,C 180,E1 -12113.925,E2 -12113.925} C_VEL
LIN {X 0,Y 515.507,Z 490.169,A -85,B 0,C 180,E1 -12113.991,E2 -12113.991} C_VEL
LIN {X 0,Y 511.4,Z 563.586,A -85,B 0,C 180,E1 -12115.404,E2 -12115.404} C_VEL
LIN {X 0,Y 507.033,Z 634.713,A -85,B 0,C 180,E1 -12116.974,E2 -12116.974} C_VEL
LIN {X 0,Y 505.734,Z 660.074,A -85,B 0,C 180,E1 -12117.682,E2 -12117.682} C_VEL
LIN {X 0,Y 504.192,Z 681.993,A -85,B 0,C 180,E1 -12118.513,E2 -12118.513} C_VEL
LIN {X 0,Y 502.295,Z 703.148,A -85,B 0,C 180,E1 -12119.537,E2 -12119.537} C_VEL
LIN {X 0,Y 500.238,Z 722.454,A -85,B 0,C 180,E1 -12120.678,E2 -12120.678} C_VEL
LIN {X 0,Y 497.916,Z 741.578,A -85,B 0,C 180,E1 -12122.037,E2 -12122.037} C_VEL
LIN {X 0,Y 495.319,Z 760.847,A -85,B 0,C 180,E1 -12123.676,E2 -12123.676} C_VEL
LIN {X 0,Y 492.74,Z 778.685,A -85,B 0,C 180,E1 -12125.482,E2 -12125.482} C_VEL
LIN {X 0,Y 490.405,Z 794.185,A -85,B 0,C 180,E1 -12127.334,E2 -12127.334} C_VEL
LIN {X 0,Y 488.202,Z 808.74,A -85,B 0,C 180,E1 -12129.373,E2 -12129.373} C_VEL
LIN {X 0,Y 486.252,Z 821.862,A -85,B 0,C 180,E1 -12131.538,E2 -12131.538} C_VEL
LIN {X 0,Y 484.599,Z 833.539,A -85,B 0,C 180,E1 -12133.826,E2 -12133.826} C_VEL
LIN {X 0,Y 483.344,Z 843.311,A -85,B 0,C 180,E1 -12136.115,E2 -12136.115} C_VEL
LIN {X 0,Y 482.33,Z 852.187,A -85,B 0,C 180,E1 -12138.682,E2 -12138.682} C_VEL
LIN {X 0,Y 481.668,Z 858.843,A -85,B 0,C 180,E1 -12141.163,E2 -12141.163} C_VEL
LIN {X 0,Y 481.264,Z 863.864,A -85,B 0,C 180,E1 -12143.678,E2 -12143.678} C_VEL
LIN {X 0,Y 481.043,Z 867.331,A -85,B 0,C 180,E1 -12146.305,E2 -12146.305} C_VEL
LIN {X 0,Y 480.959,Z 868.969,A -85,B 0,C 180,E1 -12148.69,E2 -12148.69} C_VEL
LIN {X 0,Y 480.949,Z 869.03,A -85,B 0,C 180,E1 -12151.072,E2 -12151.072} C_VEL
LIN {X 0,Y 481.028,Z 867.529,A -85,B 0,C 180,E1 -12153.575,E2 -12153.575} C_VEL
LIN {X 0,Y 481.221,Z 864.628,A -85,B 0,C 180,E1 -12155.963,E2 -12155.963} C_VEL
LIN {X 0,Y 481.579,Z 859.91,A -85,B 0,C 180,E1 -12158.477,E2 -12158.477} C_VEL
LIN {X 0,Y 482.151,Z 853.726,A -85,B 0,C 180,E1 -12160.878,E2 -12160.878} C_VEL
LIN {X 0,Y 483.082,Z 845.426,A -85,B 0,C 180,E1 -12163.404,E2 -12163.404} C_VEL
LIN {X 0,Y 484.352,Z 835.486,A -85,B 0,C 180,E1 -12165.843,E2 -12165.843} C_VEL
LIN {X 0,Y 485.91,Z 824.386,A -85,B 0,C 180,E1 -12168.103,E2 -12168.103} C_VEL
LIN {X 0,Y 487.781,Z 811.751,A -85,B 0,C 180,E1 -12170.269,E2 -12170.269} C_VEL
LIN {X 0,Y 490.049,Z 796.719,A -85,B 0,C 180,E1 -12172.437,E2 -12172.437} C_VEL
LIN {X 0,Y 492.448,Z 780.749,A -85,B 0,C 180,E1 -12174.382,E2 -12174.382} C_VEL
LIN {X 0,Y 494.892,Z 763.848,A -85,B 0,C 180,E1 -12176.133,E2 -12176.133} C_VEL
LIN {X 0,Y 497.303,Z 746.331,A -85,B 0,C 180,E1 -12177.675,E2 -12177.675} C_VEL
LIN {X 0,Y 499.687,Z 727.281,A -85,B 0,C 180,E1 -12179.094,E2 -12179.094} C_VEL
LIN {X 0,Y 501.796,Z 708.408,A -85,B 0,C 180,E1 -12180.274,E2 -12180.274} C_VEL
LIN {X 0,Y 503.782,Z 687.768,A -85,B 0,C 180,E1 -12181.333,E2 -12181.333} C_VEL
LIN {X 0,Y 505.438,Z 665.945,A -85,B 0,C 180,E1 -12182.218,E2 -12182.218} C_VEL
LIN {X 0,Y 506.645,Z 643.674,A -85,B 0,C 180,E1 -12182.899,E2 -12182.899} C_VEL
LIN {X 0,Y 509.577,Z 593.204,A -85,B 0,C 180,E1 -12184.066,E2 -12184.066} C_VEL
LIN {X 0,Y 513.995,Z 519.954,A -85,B 0,C 180,E1 -12185.554,E2 -12185.554} C_VEL
LIN {X 0,Y 517.243,Z 453.278,A -85,B 0,C 180,E1 -12186.735,E2 -12186.735} C_VEL
LIN {X 0,Y 520.245,Z 371.682,A -85,B 0,C 180,E1 -12188,E2 -12188} C_VEL
LIN {X 0,Y 523.543,Z 356.929,A -85,B 0,C 180,E1 -12188.577,E2 -12188.577} C_VEL
LIN {X 0,Y 523.906,Z 318.049,A -85,B 0,C 180,E1 -12191.239,E2 -12191.239} C_VEL
LIN {X 0,Y 523.867,Z 313.625,A -85,B 0,C 180,E1 -12191.565,E2 -12191.565} C_VEL
LIN {X 0,Y 516.028,Z 292.446,A -85,B 0,C 180,E1 -12194.077,E2 -12194.077} C_VEL
LIN {X 0,Y 507.554,Z 272.816,A -85,B 0,C 180,E1 -12196.564,E2 -12196.564} C_VEL
LIN {X 0,Y 499.437,Z 256.421,A -85,B 0,C 180,E1 -12198.83,E2 -12198.83} C_VEL
LIN {X 0,Y 492.888,Z 244.232,A -85,B 0,C 180,E1 -12200.616,E2 -12200.616} C_VEL
LIN {X 0,Y 487.544,Z 235.054,A -85,B 0,C 180,E1 -12202.029,E2 -12202.029} C_VEL
LIN {X 0,Y 485.446,Z 231.607,A -85,B 0,C 180,E1 -12202.582,E2 -12202.582} C_VEL
LIN {X 0,Y 484.643,Z 230.133,A -85,B 0,C 180,E1 -12202.807,E2 -12202.807} C_VEL
LIN {X 0,Y 482.495,Z 227.01,A -85,B 0,C 180,E1 -12203.356,E2 -12203.356} C_VEL
LIN {X 0,Y 482.043,Z 225.162,A -85,B 0,C 180,E1 -12203.593,E2 -12203.593} C_VEL
LIN {X 0,Y 482.035,Z 225.158,A -85,B 0,C 180,E1 -12207.221,E2 -12207.221} C_VEL
LIN {X 0,Y 482.048,Z 225.158,A -85,B 0,C 180,E1 -12210.84,E2 -12210.84} C_VEL
LIN {X 0,Y 482.049,Z 225.181,A -85,B 0,C 180,E1 -12214.462,E2 -12214.462} C_VEL
LIN {X 0,Y 482.044,Z 225.166,A -85,B 0,C 180,E1 -12218.076,E2 -12218.076} C_VEL
LIN {X 0,Y 482.045,Z 225.143,A -85,B 0,C 180,E1 -12221.622,E2 -12221.622} C_VEL
LIN {X 0,Y 482.048,Z 225.182,A -85,B 0,C 180,E1 -12225.218,E2 -12225.218} C_VEL
LIN {X 0,Y 482.045,Z 225.151,A -85,B 0,C 180,E1 -12228.877,E2 -12228.877} C_VEL
LIN {X 0,Y 482.033,Z 225.163,A -85,B 0,C 180,E1 -12232.491,E2 -12232.491} C_VEL
LIN {X 0,Y 482.037,Z 225.172,A -85,B 0,C 180,E1 -12236.146,E2 -12236.146} C_VEL
LIN {X 0,Y 482.053,Z 225.141,A -85,B 0,C 180,E1 -12239.762,E2 -12239.762} C_VEL
LIN {X 0,Y 482.05,Z 225.182,A -85,B 0,C 180,E1 -12243.449,E2 -12243.449} C_VEL
LIN {X 0,Y 482.056,Z 225.134,A -85,B 0,C 180,E1 -12247.149,E2 -12247.149} C_VEL
LIN {X 0,Y 482.032,Z 225.185,A -85,B 0,C 180,E1 -12250.76,E2 -12250.76} C_VEL
LIN {X 0,Y 482.025,Z 225.184,A -85,B 0,C 180,E1 -12254.414,E2 -12254.414} C_VEL
LIN {X 0,Y 482.04,Z 225.178,A -85,B 0,C 180,E1 -12258.003,E2 -12258.003} C_VEL
LIN {X 0,Y 482.059,Z 225.174,A -85,B 0,C 180,E1 -12261.539,E2 -12261.539} C_VEL
LIN {X 0,Y 482.04,Z 225.184,A -85,B 0,C 180,E1 -12265.165,E2 -12265.165} C_VEL
LIN {X 0,Y 482.032,Z 225.293,A -85,B 0,C 180,E1 -12268.515,E2 -12268.515} C_VEL
LIN {X 0,Y 483.413,Z 228.767,A -85,B 0,C 180,E1 -12269.083,E2 -12269.083} C_VEL
LIN {X 0,Y 484.613,Z 230.742,A -85,B 0,C 180,E1 -12269.46,E2 -12269.46} C_VEL
LIN {X 0,Y 491.59,Z 244.301,A -85,B 0,C 180,E1 -12271.79,E2 -12271.79} C_VEL
LIN {X 0,Y 501.162,Z 263.07,A -85,B 0,C 180,E1 -12274.793,E2 -12274.793} C_VEL
LIN {X 0,Y 510.817,Z 282.52,A -85,B 0,C 180,E1 -12277.642,E2 -12277.642} C_VEL
LIN {X 0,Y 521.719,Z 305.144,A -85,B 0,C 180,E1 -12280.664,E2 -12280.664} C_VEL
LIN {X 0,Y 527.639,Z 317.579,A -85,B 0,C 180,E1 -12282.169,E2 -12282.169} C_VEL
LIN {X 0,Y 528.388,Z 319.377,A -85,B 0,C 180,E1 -12282.272,E2 -12282.272} C_VEL
LIN {X 0,Y 530.976,Z 346.541,A -85,B 0,C 180,E1 -12283.057,E2 -12283.057} C_VEL
LIN {X 0,Y 520.798,Z 584.167,A -85,B 0,C 180,E1 -12286.965,E2 -12286.965} C_VEL
LIN {X 0,Y 516.743,Z 692.909,A -85,B 0,C 180,E1 -12288.729,E2 -12288.729} C_VEL
LIN {X 0,Y 514.996,Z 717.542,A -85,B 0,C 180,E1 -12289.312,E2 -12289.312} C_VEL
LIN {X 0,Y 512.9,Z 741.527,A -85,B 0,C 180,E1 -12290.065,E2 -12290.065} C_VEL
LIN {X 0,Y 510.48,Z 763.973,A -85,B 0,C 180,E1 -12290.97,E2 -12290.97} C_VEL
LIN {X 0,Y 507.695,Z 786.913,A -85,B 0,C 180,E1 -12292.086,E2 -12292.086} C_VEL
LIN {X 0,Y 504.938,Z 807.104,A -85,B 0,C 180,E1 -12293.271,E2 -12293.271} C_VEL
LIN {X 0,Y 501.736,Z 828.946,A -85,B 0,C 180,E1 -12294.765,E2 -12294.765} C_VEL
LIN {X 0,Y 498.725,Z 848.133,A -85,B 0,C 180,E1 -12296.308,E2 -12296.308} C_VEL
LIN {X 0,Y 495.535,Z 868.127,A -85,B 0,C 180,E1 -12298.157,E2 -12298.157} C_VEL
LIN {X 0,Y 492.721,Z 885.167,A -85,B 0,C 180,E1 -12299.985,E2 -12299.985} C_VEL
LIN {X 0,Y 489.866,Z 902.698,A -85,B 0,C 180,E1 -12302.133,E2 -12302.133} C_VEL
LIN {X 0,Y 487.535,Z 917.493,A -85,B 0,C 180,E1 -12304.228,E2 -12304.228} C_VEL
LIN {X 0,Y 485.38,Z 932.046,A -85,B 0,C 180,E1 -12306.573,E2 -12306.573} C_VEL
LIN {X 0,Y 483.617,Z 945.097,A -85,B 0,C 180,E1 -12309.042,E2 -12309.042} C_VEL
LIN {X 0,Y 482.24,Z 956.932,A -85,B 0,C 180,E1 -12311.63,E2 -12311.63} C_VEL
LIN {X 0,Y 481.315,Z 966.481,A -85,B 0,C 180,E1 -12314.122,E2 -12314.122} C_VEL
LIN {X 0,Y 480.711,Z 975.059,A -85,B 0,C 180,E1 -12316.773,E2 -12316.773} C_VEL
LIN {X 0,Y 480.38,Z 982.148,A -85,B 0,C 180,E1 -12319.567,E2 -12319.567} C_VEL
LIN {X 0,Y 480.277,Z 986.95,A -85,B 0,C 180,E1 -12321.982,E2 -12321.982} C_VEL
LIN {X 0,Y 480.276,Z 990.842,A -85,B 0,C 180,E1 -12324.744,E2 -12324.744} C_VEL
LIN {X 0,Y 480.325,Z 992.832,A -85,B 0,C 180,E1 -12327.136,E2 -12327.136} C_VEL
LIN {X 0,Y 480.359,Z 993.6,A -85,B 0,C 180,E1 -12329.404,E2 -12329.404} C_VEL
LIN {X 0,Y 480.373,Z 993.062,A -85,B 0,C 180,E1 -12332.147,E2 -12332.147} C_VEL
LIN {X 0,Y 480.341,Z 991.019,A -85,B 0,C 180,E1 -12334.657,E2 -12334.657} C_VEL
LIN {X 0,Y 480.333,Z 988.012,A -85,B 0,C 180,E1 -12336.935,E2 -12336.935} C_VEL
LIN {X 0,Y 480.399,Z 982.868,A -85,B 0,C 180,E1 -12339.706,E2 -12339.706} C_VEL
LIN {X 0,Y 480.63,Z 976.14,A -85,B 0,C 180,E1 -12342.373,E2 -12342.373} C_VEL
LIN {X 0,Y 481.098,Z 968.23,A -85,B 0,C 180,E1 -12344.935,E2 -12344.935} C_VEL
LIN {X 0,Y 481.928,Z 958.026,A -85,B 0,C 180,E1 -12347.633,E2 -12347.633} C_VEL
LIN {X 0,Y 483.045,Z 947.101,A -85,B 0,C 180,E1 -12350.097,E2 -12350.097} C_VEL
LIN {X 0,Y 484.741,Z 933.138,A -85,B 0,C 180,E1 -12352.773,E2 -12352.773} C_VEL
LIN {X 0,Y 486.733,Z 918.717,A -85,B 0,C 180,E1 -12355.166,E2 -12355.166} C_VEL
LIN {X 0,Y 489.164,Z 902.254,A -85,B 0,C 180,E1 -12357.514,E2 -12357.514} C_VEL
LIN {X 0,Y 491.937,Z 884.819,A -85,B 0,C 180,E1 -12359.694,E2 -12359.694} C_VEL
LIN {X 0,Y 494.968,Z 865.802,A -85,B 0,C 180,E1 -12361.737,E2 -12361.737} C_VEL
LIN {X 0,Y 498.219,Z 845.5,A -85,B 0,C 180,E1 -12363.636,E2 -12363.636} C_VEL
LIN {X 0,Y 501.361,Z 825.535,A -85,B 0,C 180,E1 -12365.243,E2 -12365.243} C_VEL
LIN {X 0,Y 504.856,Z 802.069,A -85,B 0,C 180,E1 -12366.856,E2 -12366.856} C_VEL
LIN {X 0,Y 508.054,Z 779.456,A -85,B 0,C 180,E1 -12368.169,E2 -12368.169} C_VEL
LIN {X 0,Y 511.015,Z 755.84,A -85,B 0,C 180,E1 -12369.29,E2 -12369.29} C_VEL
LIN {X 0,Y 513.846,Z 730.482,A -85,B 0,C 180,E1 -12370.259,E2 -12370.259} C_VEL
LIN {X 0,Y 516.054,Z 707.13,A -85,B 0,C 180,E1 -12370.953,E2 -12370.953} C_VEL
LIN {X 0,Y 517.709,Z 682.779,A -85,B 0,C 180,E1 -12371.48,E2 -12371.48} C_VEL
LIN {X 0,Y 522.492,Z 593.531,A -85,B 0,C 180,E1 -12373.079,E2 -12373.079} C_VEL
LIN {X 0,Y 527.819,Z 522.285,A -85,B 0,C 180,E1 -12374.482,E2 -12374.482} C_VEL
LIN {X 0,Y 534.576,Z 454.884,A -85,B 0,C 180,E1 -12375.925,E2 -12375.925} C_VEL
LIN {X 0,Y 542.768,Z 392.347,A -85,B 0,C 180,E1 -12377.325,E2 -12377.325} C_VEL
LIN {X 0,Y 548.127,Z 358.958,A -85,B 0,C 180,E1 -12378.097,E2 -12378.097} C_VEL
LIN {X 0,Y 550.284,Z 355.693,A -85,B 0,C 180,E1 -12378.245,E2 -12378.245} C_VEL
LIN {X 0,Y 544.284,Z 365.012,A -85,B 0,C 180,E1 -12379.312,E2 -12379.312} C_VEL
LIN {X 0,Y 539.398,Z 380.968,A -85,B 0,C 180,E1 -12380.879,E2 -12380.879} C_VEL
LIN {X 0,Y 536.467,Z 395.147,A -85,B 0,C 180,E1 -12382.127,E2 -12382.127} C_VEL
LIN {X 0,Y 533.779,Z 414.563,A -85,B 0,C 180,E1 -12383.63,E2 -12383.63} C_VEL
LIN {X 0,Y 531.595,Z 437.999,A -85,B 0,C 180,E1 -12385.173,E2 -12385.173} C_VEL
LIN {X 0,Y 529.823,Z 465.535,A -85,B 0,C 180,E1 -12386.737,E2 -12386.737} C_VEL
LIN {X 0,Y 528.165,Z 497.407,A -85,B 0,C 180,E1 -12388.284,E2 -12388.284} C_VEL
LIN {X 0,Y 527.364,Z 510.645,A -85,B 0,C 180,E1 -12388.84,E2 -12388.84} C_VEL
LIN {X 0,Y 513.633,Z 618.773,A -85,B 0,C 180,E1 -12391.728,E2 -12391.728} C_VEL
LIN {X 0,Y 505.897,Z 692.84,A -85,B 0,C 180,E1 -12393.755,E2 -12393.755} C_VEL
LIN {X 0,Y 503.288,Z 716.231,A -85,B 0,C 180,E1 -12394.619,E2 -12394.619} C_VEL
LIN {X 0,Y 500.643,Z 739.505,A -85,B 0,C 180,E1 -12395.705,E2 -12395.705} C_VEL
LIN {X 0,Y 497.962,Z 761.93,A -85,B 0,C 180,E1 -12397.011,E2 -12397.011} C_VEL
LIN {X 0,Y 495.654,Z 780.628,A -85,B 0,C 180,E1 -12398.336,E2 -12398.336} C_VEL
LIN {X 0,Y 493.5,Z 797.932,A -85,B 0,C 180,E1 -12399.79,E2 -12399.79} C_VEL
LIN {X 0,Y 491.299,Z 814.753,A -85,B 0,C 180,E1 -12401.489,E2 -12401.489} C_VEL
LIN {X 0,Y 489.46,Z 828.363,A -85,B 0,C 180,E1 -12403.137,E2 -12403.137} C_VEL
LIN {X 0,Y 487.778,Z 840.637,A -85,B 0,C 180,E1 -12404.91,E2 -12404.91} C_VEL
LIN {X 0,Y 486.254,Z 851.38,A -85,B 0,C 180,E1 -12406.806,E2 -12406.806} C_VEL
LIN {X 0,Y 485,Z 860.123,A -85,B 0,C 180,E1 -12408.705,E2 -12408.705} C_VEL
LIN {X 0,Y 483.928,Z 867.372,A -85,B 0,C 180,E1 -12410.726,E2 -12410.726} C_VEL
LIN {X 0,Y 483.068,Z 873.043,A -85,B 0,C 180,E1 -12412.866,E2 -12412.866} C_VEL
LIN {X 0,Y 482.428,Z 876.766,A -85,B 0,C 180,E1 -12415.006,E2 -12415.006} C_VEL
LIN {X 0,Y 481.978,Z 878.679,A -85,B 0,C 180,E1 -12417.146,E2 -12417.146} C_VEL
LIN {X 0,Y 481.691,Z 878.819,A -85,B 0,C 180,E1 -12419.286,E2 -12419.286} C_VEL
LIN {X 0,Y 481.53,Z 877.212,A -85,B 0,C 180,E1 -12421.428,E2 -12421.428} C_VEL
LIN {X 0,Y 481.494,Z 873.875,A -85,B 0,C 180,E1 -12423.572,E2 -12423.572} C_VEL
LIN {X 0,Y 481.605,Z 868.768,A -85,B 0,C 180,E1 -12425.719,E2 -12425.719} C_VEL
LIN {X 0,Y 481.881,Z 861.783,A -85,B 0,C 180,E1 -12427.871,E2 -12427.871} C_VEL
LIN {X 0,Y 482.339,Z 853.305,A -85,B 0,C 180,E1 -12429.908,E2 -12429.908} C_VEL
LIN {X 0,Y 483.039,Z 842.79,A -85,B 0,C 180,E1 -12431.947,E2 -12431.947} C_VEL
LIN {X 0,Y 483.945,Z 830.754,A -85,B 0,C 180,E1 -12433.867,E2 -12433.867} C_VEL
LIN {X 0,Y 485.074,Z 816.864,A -85,B 0,C 180,E1 -12435.712,E2 -12435.712} C_VEL
LIN {X 0,Y 486.362,Z 801.625,A -85,B 0,C 180,E1 -12437.405,E2 -12437.405} C_VEL
LIN {X 0,Y 487.79,Z 784.779,A -85,B 0,C 180,E1 -12438.968,E2 -12438.968} C_VEL
LIN {X 0,Y 489.22,Z 767.155,A -85,B 0,C 180,E1 -12440.332,E2 -12440.332} C_VEL
LIN {X 0,Y 490.684,Z 748.607,A -85,B 0,C 180,E1 -12441.518,E2 -12441.518} C_VEL
LIN {X 0,Y 492.088,Z 729.343,A -85,B 0,C 180,E1 -12442.521,E2 -12442.521} C_VEL
LIN {X 0,Y 493.436,Z 708.088,A -85,B 0,C 180,E1 -12443.387,E2 -12443.387} C_VEL
LIN {X 0,Y 494.621,Z 686.149,A -85,B 0,C 180,E1 -12444.046,E2 -12444.046} C_VEL
LIN {X 0,Y 496.191,Z 644.603,A -85,B 0,C 180,E1 -12444.88,E2 -12444.88} C_VEL
LIN {X 0,Y 501.976,Z 499.387,A -85,B 0,C 180,E1 -12447.671,E2 -12447.671} C_VEL
LIN {X 0,Y 497.08,Z 445.289,A -85,B 0,C 180,E1 -12449.19,E2 -12449.19} C_VEL
LIN {X 0,Y 501.552,Z 393.19,A -85,B 0,C 180,E1 -12453.042,E2 -12453.042} C_VEL
LIN {X 0,Y 506.339,Z 343.384,A -85,B 0,C 180,E1 -12456.752,E2 -12456.752} C_VEL
LIN {X 0,Y 511.134,Z 297.518,A -85,B 0,C 180,E1 -12460.199,E2 -12460.199} C_VEL
LIN {X 0,Y 502.711,Z 274.81,A -85,B 0,C 180,E1 -12462.862,E2 -12462.862} C_VEL
LIN {X 0,Y 502.414,Z 273.908,A -85,B 0,C 180,E1 -12462.993,E2 -12462.993} C_VEL
LIN {X 0,Y 504.462,Z 274.528,A -85,B 0,C 180,E1 -12463.299,E2 -12463.299} C_VEL
LIN {X 0,Y 508.475,Z 274.849,A -85,B 0,C 180,E1 -12463.806,E2 -12463.806} C_VEL
LIN {X 0,Y 516.549,Z 293.957,A -85,B 0,C 180,E1 -12466.222,E2 -12466.222} C_VEL
LIN {X 0,Y 523.91,Z 313.859,A -85,B 0,C 180,E1 -12468.568,E2 -12468.568} C_VEL
LIN {X 0,Y 523.449,Z 356.947,A -85,B 0,C 180,E1 -12471.528,E2 -12471.528} C_VEL
LIN {X 0,Y 519.968,Z 373.528,A -85,B 0,C 180,E1 -12472.147,E2 -12472.147} C_VEL
LIN {X 0,Y 516.931,Z 459.567,A -85,B 0,C 180,E1 -12473.463,E2 -12473.463} C_VEL
LIN {X 0,Y 515.507,Z 490.169,A -85,B 0,C 180,E1 -12473.991,E2 -12473.991} C_VEL
LIN {X 0,Y 514.345,Z 497.819,A -85,B 0,C 180,E1 -12474.062,E2 -12474.062} C_VEL
LIN {X 0,Y 508.267,Z 518.177,A -85,B 0,C 180,E1 -12474.017,E2 -12474.017} C_VEL
LIN {X 0,Y 507.289,Z 524.733,A -85,B 0,C 180,E1 -12474.092,E2 -12474.092} C_VEL
LIN {X 0,Y 502.493,Z 600.764,A -85,B 0,C 180,E1 -12475.674,E2 -12475.674} C_VEL
LIN {X 0,Y 499.772,Z 646.534,A -85,B 0,C 180,E1 -12476.77,E2 -12476.77} C_VEL
